Yaskawa INFORM job: DEMO_ROOF_UPPER_0625_3PAINT_32.JBI

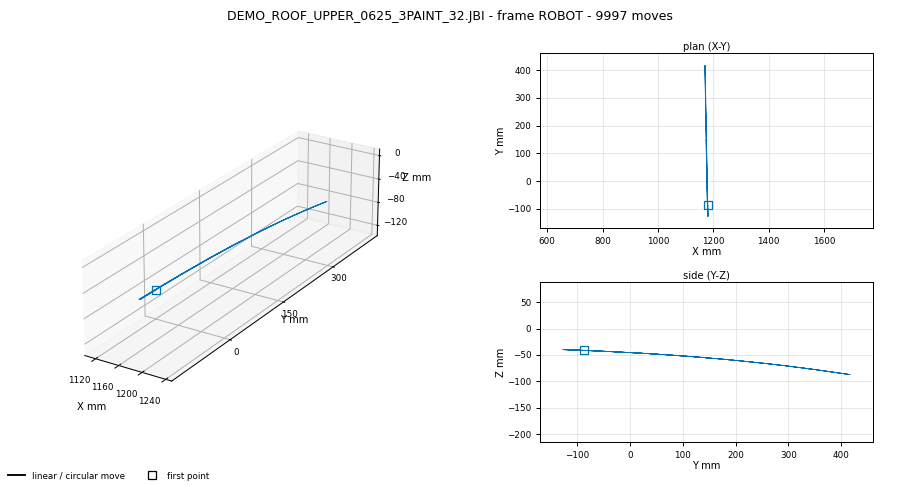
[picture p0: tool path of DEMO_ROOF_UPPER_0625_3PAINT_32.JBI in frame ROBOT, 9997 of 9997 moves have a stored position in this frame; points joined in program order, loops and branches not executed]
/JOB
//NAME DEMO_ROOF_UPPER_0625_3PAINT32
//POS
///NPOS 9997,0,0,0,0,0
///TOOL 0
///USER 0
///POSTYPE ROBOT
///RECTAN
///RCONF 1,0,0,0,0,0,0,0,0,0,0,0,0,0,0,0,0,0,0,0,0,0,0,0
C00000=1180.543,-86.813,-41.166,179.183,5.706,149.254
C00001=1180.548,-87.062,-41.157,179.181,5.706,149.255
C00002=1180.554,-87.312,-41.146,179.179,5.706,149.256
C00003=1180.559,-87.563,-41.136,179.177,5.705,149.256
C00004=1180.565,-87.812,-41.126,179.174,5.706,149.257
C00005=1180.570,-88.062,-41.116,179.172,5.705,149.257
C00006=1180.574,-88.312,-41.106,179.170,5.705,149.258
C00007=1180.580,-88.561,-41.096,179.168,5.704,149.259
C00008=1180.586,-88.811,-41.086,179.165,5.704,149.259
C00009=1180.591,-89.061,-41.075,179.163,5.704,149.260
C00010=1180.596,-89.310,-41.065,179.161,5.704,149.260
C00011=1180.601,-89.560,-41.055,179.159,5.704,149.261
C00012=1180.607,-89.809,-41.045,179.157,5.703,149.262
C00013=1180.612,-90.060,-41.035,179.154,5.703,149.262
C00014=1180.617,-90.310,-41.026,179.153,5.703,149.263
C00015=1180.622,-90.559,-41.015,179.150,5.702,149.264
C00016=1180.627,-90.809,-41.005,179.148,5.703,149.264
C00017=1180.633,-91.059,-40.995,179.146,5.702,149.265
C00018=1180.638,-91.308,-40.985,179.143,5.703,149.265
C00019=1180.644,-91.558,-40.975,179.141,5.702,149.266
C00020=1180.649,-91.809,-40.965,179.139,5.701,149.267
C00021=1180.654,-92.058,-40.955,179.137,5.701,149.267
C00022=1180.659,-92.307,-40.945,179.134,5.701,149.268
C00023=1180.665,-92.557,-40.935,179.132,5.701,149.269
C00024=1180.669,-92.807,-40.925,179.130,5.701,149.269
C00025=1180.675,-93.057,-40.915,179.127,5.700,149.270
C00026=1180.681,-93.307,-40.905,179.126,5.700,149.270
C00027=1180.686,-93.556,-40.896,179.123,5.700,149.271
C00028=1180.691,-93.806,-40.885,179.122,5.700,149.271
C00029=1180.696,-94.056,-40.876,179.119,5.699,149.272
C00030=1180.701,-94.305,-40.866,179.117,5.699,149.273
C00031=1180.707,-94.555,-40.856,179.115,5.699,149.273
C00032=1180.712,-94.804,-40.845,179.112,5.699,149.274
C00033=1180.717,-95.055,-40.836,179.110,5.699,149.275
C00034=1180.723,-95.305,-40.826,179.108,5.698,149.275
C00035=1180.728,-95.554,-40.816,179.106,5.698,149.276
C00036=1180.733,-95.803,-40.806,179.103,5.698,149.276
C00037=1180.739,-96.054,-40.797,179.102,5.698,149.277
C00038=1180.744,-96.304,-40.786,179.099,5.697,149.278
C00039=1180.749,-96.553,-40.777,179.097,5.697,149.278
C00040=1180.755,-96.803,-40.767,179.095,5.697,149.279
C00041=1180.760,-97.052,-40.757,179.092,5.697,149.280
C00042=1180.765,-97.302,-40.747,179.091,5.697,149.280
C00043=1180.771,-97.553,-40.737,179.088,5.696,149.281
C00044=1180.775,-97.802,-40.728,179.086,5.696,149.281
C00045=1180.781,-98.052,-40.718,179.084,5.696,149.282
C00046=1180.786,-98.301,-40.709,179.081,5.695,149.282
C00047=1180.792,-98.551,-40.698,179.079,5.696,149.283
C00048=1180.797,-98.800,-40.688,179.077,5.695,149.284
C00049=1180.802,-99.051,-40.679,179.075,5.695,149.284
C00050=1180.808,-99.301,-40.669,179.073,5.694,149.285
C00051=1180.813,-99.550,-40.660,179.071,5.695,149.285
C00052=1180.818,-99.800,-40.650,179.069,5.694,149.286
C00053=1180.823,-100.049,-40.640,179.066,5.694,149.287
C00054=1180.829,-100.299,-40.631,179.064,5.694,149.287
C00055=1180.834,-100.549,-40.621,179.062,5.693,149.288
C00056=1180.839,-100.799,-40.611,179.060,5.694,149.289
C00057=1180.844,-101.049,-40.601,179.057,5.693,149.289
C00058=1180.850,-101.298,-40.591,179.055,5.693,149.290
C00059=1180.855,-101.570,-40.581,179.053,5.692,149.290
C00060=1180.861,-101.841,-40.571,179.050,5.692,149.291
C00061=1180.868,-102.114,-40.560,179.048,5.692,149.292
C00062=1180.873,-102.385,-40.549,179.046,5.692,149.292
C00063=1180.879,-102.635,-40.540,179.043,5.691,149.293
C00064=1180.883,-102.884,-40.530,179.041,5.692,149.294
C00065=1180.889,-103.134,-40.521,179.039,5.691,149.294
C00066=1180.894,-103.384,-40.511,179.037,5.691,149.295
C00067=1180.899,-103.634,-40.502,179.035,5.691,149.295
C00068=1180.904,-103.884,-40.492,179.033,5.691,149.296
C00069=1180.910,-104.134,-40.483,179.031,5.690,149.297
C00070=1180.915,-104.383,-40.473,179.029,5.691,149.297
C00071=1180.920,-104.633,-40.464,179.026,5.690,149.298
C00072=1180.926,-104.883,-40.453,179.024,5.689,149.298
C00073=1180.931,-105.132,-40.445,179.022,5.689,149.299
C00074=1180.937,-105.383,-40.435,179.019,5.689,149.300
C00075=1180.942,-105.632,-40.425,179.018,5.689,149.300
C00076=1180.947,-105.882,-40.417,179.015,5.689,149.301
C00077=1180.953,-106.131,-40.406,179.014,5.689,149.301
C00078=1180.957,-106.382,-40.397,179.011,5.688,149.302
C00079=1180.963,-106.631,-40.387,179.009,5.688,149.303
C00080=1180.968,-106.881,-40.378,179.007,5.688,149.303
C00081=1180.974,-107.131,-40.368,179.005,5.688,149.304
C00082=1180.979,-107.381,-40.359,179.002,5.688,149.304
C00083=1180.984,-107.630,-40.350,179.001,5.688,149.305
C00084=1180.989,-107.880,-40.340,178.998,5.687,149.306
C00085=1180.995,-108.130,-40.331,178.996,5.686,149.306
C00086=1181.000,-108.380,-40.322,178.994,5.687,149.307
C00087=1181.005,-108.629,-40.312,178.992,5.686,149.307
C00088=1181.011,-108.879,-40.303,178.989,5.686,149.308
C00089=1181.016,-109.129,-40.293,178.987,5.686,149.309
C00090=1181.021,-109.378,-40.284,178.985,5.686,149.309
C00091=1181.026,-109.628,-40.275,178.983,5.685,149.310
C00092=1181.032,-109.878,-40.265,178.981,5.686,149.310
C00093=1181.037,-110.128,-40.256,178.979,5.685,149.311
C00094=1181.042,-110.378,-40.247,178.977,5.685,149.312
C00095=1181.048,-110.627,-40.237,178.974,5.685,149.312
C00096=1181.053,-110.877,-40.228,178.972,5.685,149.313
C00097=1181.058,-111.127,-40.219,178.970,5.684,149.313
C00098=1181.064,-111.377,-40.209,178.968,5.685,149.314
C00099=1181.069,-111.626,-40.200,178.966,5.684,149.314
C00100=1181.074,-111.876,-40.191,178.964,5.684,149.315
C00101=1181.080,-112.126,-40.181,178.962,5.683,149.316
C00102=1181.085,-112.375,-40.172,178.960,5.684,149.316
C00103=1181.090,-112.625,-40.163,178.957,5.683,149.317
C00104=1181.096,-112.875,-40.153,178.955,5.683,149.318
C00105=1181.101,-113.125,-40.144,178.953,5.683,149.318
C00106=1181.106,-113.375,-40.135,178.950,5.682,149.319
C00107=1181.111,-113.624,-40.126,178.949,5.682,149.319
C00108=1181.117,-113.875,-40.116,178.946,5.682,149.320
C00109=1181.122,-114.124,-40.108,178.945,5.682,149.320
C00110=1181.128,-114.374,-40.099,178.942,5.682,149.321
C00111=1181.133,-114.624,-40.088,178.940,5.682,149.322
C00112=1181.138,-114.874,-40.080,178.938,5.681,149.322
C00113=1181.143,-115.124,-40.071,178.936,5.681,149.323
C00114=1181.149,-115.373,-40.062,178.934,5.680,149.323
C00115=1181.155,-115.624,-40.052,178.932,5.681,149.324
C00116=1181.159,-115.873,-40.043,178.930,5.680,149.325
C00117=1181.165,-116.123,-40.034,178.927,5.681,149.325
C00118=1181.170,-116.372,-40.025,178.925,5.680,149.326
C00119=1181.176,-116.622,-40.016,178.923,5.680,149.327
C00120=1181.181,-116.872,-40.007,178.921,5.679,149.327
C00121=1181.187,-117.122,-39.998,178.919,5.680,149.328
C00122=1181.191,-117.371,-39.988,178.917,5.679,149.328
C00123=1181.197,-117.621,-39.979,178.915,5.679,149.329
C00124=1181.203,-117.871,-39.970,178.912,5.679,149.329
C00125=1181.208,-118.121,-39.961,178.911,5.679,149.330
C00126=1181.213,-118.371,-39.952,178.908,5.678,149.331
C00127=1181.218,-118.620,-39.943,178.907,5.678,149.331
C00128=1181.223,-118.870,-39.934,178.904,5.678,149.332
C00129=1181.229,-119.120,-39.925,178.902,5.678,149.332
C00130=1181.235,-119.369,-39.916,178.900,5.678,149.333
C00131=1181.240,-119.619,-39.907,178.898,5.678,149.333
C00132=1181.245,-119.869,-39.898,178.895,5.677,149.334
C00133=1181.250,-120.119,-39.889,178.894,5.677,149.335
C00134=1181.255,-120.368,-39.880,178.892,5.676,149.335
C00135=1181.261,-120.619,-39.870,178.889,5.677,149.336
C00136=1181.266,-120.868,-39.862,178.887,5.676,149.336
C00137=1181.271,-121.118,-39.853,178.885,5.677,149.337
C00138=1181.277,-121.368,-39.844,178.883,5.676,149.338
C00139=1181.282,-121.617,-39.835,178.881,5.676,149.338
C00140=1181.288,-121.867,-39.826,178.879,5.675,149.339
C00141=1181.293,-122.117,-39.817,178.877,5.676,149.339
C00142=1181.299,-122.367,-39.808,178.874,5.675,149.340
C00143=1181.304,-122.617,-39.799,178.873,5.675,149.340
C00144=1181.309,-122.867,-39.790,178.870,5.675,149.341
C00145=1181.314,-123.117,-39.781,178.869,5.675,149.342
C00146=1181.320,-123.366,-39.773,178.866,5.674,149.342
C00147=1181.325,-123.616,-39.764,178.864,5.674,149.343
C00148=1181.330,-123.866,-39.755,178.862,5.675,149.344
C00149=1181.335,-124.115,-39.746,178.860,5.674,149.344
C00150=1181.341,-124.365,-39.737,178.858,5.674,149.345
C00151=1181.346,-124.615,-39.728,178.856,5.674,149.345
C00152=1181.351,-124.865,-39.719,178.854,5.674,149.346
C00153=1181.357,-125.114,-39.710,178.851,5.673,149.346
C00154=1181.363,-125.364,-39.701,178.850,5.673,149.347
C00155=1181.368,-125.614,-39.692,178.847,5.673,149.348
C00156=1181.373,-125.864,-39.684,178.846,5.673,149.348
C00157=1181.378,-126.114,-39.675,178.843,5.672,149.349
C00158=1181.384,-126.363,-39.666,178.841,5.673,149.349
C00159=1181.389,-126.613,-39.658,178.839,5.672,149.350
C00160=1181.394,-126.863,-39.649,178.837,5.672,149.351
C00161=1181.400,-127.113,-39.640,178.835,5.672,149.351
C00162=1181.405,-127.363,-39.631,178.833,5.672,149.352
C00163=1180.984,-127.374,-39.672,178.829,5.675,149.353
C00164=1180.979,-127.124,-39.681,178.831,5.675,149.353
C00165=1180.973,-126.875,-39.689,178.833,5.676,149.352
C00166=1180.967,-126.624,-39.697,178.835,5.675,149.352
C00167=1180.962,-126.374,-39.706,178.837,5.676,149.351
C00168=1180.957,-126.124,-39.715,178.839,5.675,149.351
C00169=1180.952,-125.874,-39.724,178.842,5.676,149.350
C00170=1180.946,-125.625,-39.733,178.843,5.676,149.350
C00171=1180.941,-125.376,-39.741,178.846,5.677,149.349
C00172=1180.936,-125.126,-39.750,178.847,5.677,149.348
C00173=1180.931,-124.876,-39.759,178.850,5.677,149.348
C00174=1180.925,-124.626,-39.768,178.852,5.677,149.347
C00175=1180.920,-124.376,-39.777,178.854,5.678,149.347
C00176=1180.914,-124.127,-39.786,178.856,5.677,149.346
C00177=1180.909,-123.877,-39.795,178.858,5.678,149.345
C00178=1180.903,-123.627,-39.804,178.860,5.678,149.345
C00179=1180.898,-123.377,-39.813,178.863,5.678,149.344
C00180=1180.893,-123.127,-39.822,178.865,5.678,149.344
C00181=1180.888,-122.877,-39.831,178.867,5.679,149.343
C00182=1180.883,-122.628,-39.840,178.868,5.679,149.343
C00183=1180.877,-122.378,-39.848,178.871,5.679,149.342
C00184=1180.872,-122.129,-39.857,178.873,5.679,149.341
C00185=1180.867,-121.879,-39.866,178.875,5.679,149.341
C00186=1180.861,-121.629,-39.875,178.877,5.679,149.340
C00187=1180.856,-121.379,-39.884,178.880,5.680,149.339
C00188=1180.850,-121.129,-39.893,178.881,5.680,149.339
C00189=1180.845,-120.879,-39.902,178.883,5.681,149.338
C00190=1180.839,-120.630,-39.911,178.886,5.680,149.338
C00191=1180.834,-120.380,-39.919,178.888,5.681,149.337
C00192=1180.829,-120.130,-39.928,178.890,5.680,149.337
C00193=1180.823,-119.880,-39.938,178.892,5.681,149.336
C00194=1180.818,-119.630,-39.947,178.894,5.681,149.335
C00195=1180.813,-119.380,-39.956,178.896,5.682,149.335
C00196=1180.808,-119.130,-39.965,178.898,5.681,149.334
C00197=1180.803,-118.881,-39.973,178.901,5.682,149.334
C00198=1180.798,-118.631,-39.983,178.902,5.682,149.333
C00199=1180.792,-118.381,-39.993,178.905,5.682,149.332
C00200=1180.786,-118.132,-40.001,178.906,5.682,149.332
C00201=1180.781,-117.882,-40.010,178.909,5.683,149.331
C00202=1180.776,-117.632,-40.019,178.911,5.683,149.331
C00203=1180.770,-117.382,-40.028,178.913,5.683,149.330
C00204=1180.765,-117.132,-40.037,178.915,5.683,149.330
C00205=1180.759,-116.882,-40.046,178.918,5.683,149.329
C00206=1180.755,-116.633,-40.056,178.919,5.683,149.328
C00207=1180.749,-116.383,-40.065,178.922,5.684,149.328
C00208=1180.744,-116.133,-40.074,178.924,5.684,149.327
C00209=1180.738,-115.883,-40.083,178.926,5.685,149.327
C00210=1180.733,-115.633,-40.092,178.928,5.684,149.326
C00211=1180.728,-115.384,-40.101,178.930,5.685,149.325
C00212=1180.723,-115.134,-40.110,178.932,5.684,149.325
C00213=1180.717,-114.884,-40.120,178.934,5.685,149.324
C00214=1180.711,-114.635,-40.129,178.936,5.685,149.324
C00215=1180.706,-114.385,-40.137,178.939,5.686,149.323
C00216=1180.700,-114.135,-40.147,178.941,5.685,149.322
C00217=1180.696,-113.886,-40.157,178.943,5.686,149.322
C00218=1180.690,-113.636,-40.165,178.945,5.686,149.321
C00219=1180.685,-113.386,-40.174,178.947,5.686,149.321
C00220=1180.679,-113.136,-40.184,178.949,5.686,149.320
C00221=1180.674,-112.887,-40.193,178.951,5.687,149.319
C00222=1180.669,-112.637,-40.202,178.953,5.686,149.319
C00223=1180.663,-112.387,-40.212,178.956,5.687,149.318
C00224=1180.658,-112.137,-40.221,178.957,5.687,149.318
C00225=1180.653,-111.888,-40.230,178.960,5.687,149.317
C00226=1180.648,-111.638,-40.239,178.962,5.687,149.317
C00227=1180.642,-111.388,-40.249,178.964,5.688,149.316
C00228=1180.637,-111.138,-40.258,178.966,5.688,149.315
C00229=1180.632,-110.889,-40.267,178.968,5.688,149.315
C00230=1180.626,-110.638,-40.277,178.970,5.688,149.314
C00231=1180.621,-110.389,-40.286,178.973,5.689,149.313
C00232=1180.616,-110.139,-40.295,178.974,5.689,149.313
C00233=1180.610,-109.889,-40.305,178.977,5.689,149.312
C00234=1180.605,-109.639,-40.314,178.979,5.690,149.312
C00235=1180.600,-109.390,-40.324,178.981,5.689,149.311
C00236=1180.594,-109.140,-40.333,178.984,5.690,149.311
C00237=1180.589,-108.890,-40.342,178.986,5.690,149.310
C00238=1180.584,-108.641,-40.352,178.988,5.690,149.309
C00239=1180.579,-108.391,-40.361,178.990,5.690,149.309
C00240=1180.573,-108.141,-40.370,178.992,5.691,149.308
C00241=1180.568,-107.891,-40.380,178.994,5.690,149.307
C00242=1180.563,-107.641,-40.389,178.996,5.691,149.307
C00243=1180.557,-107.392,-40.399,178.998,5.691,149.306
C00244=1180.552,-107.141,-40.408,179.001,5.692,149.306
C00245=1180.547,-106.891,-40.417,179.003,5.691,149.305
C00246=1180.542,-106.642,-40.427,179.005,5.692,149.305
C00247=1180.536,-106.392,-40.436,179.007,5.691,149.304
C00248=1180.531,-106.143,-40.446,179.009,5.692,149.303
C00249=1180.526,-105.893,-40.455,179.012,5.693,149.303
C00250=1180.521,-105.643,-40.465,179.013,5.693,149.302
C00251=1180.515,-105.393,-40.474,179.016,5.693,149.301
C00252=1180.510,-105.143,-40.483,179.018,5.693,149.301
C00253=1180.504,-104.894,-40.494,179.020,5.693,149.300
C00254=1180.499,-104.644,-40.502,179.022,5.693,149.300
C00255=1180.493,-104.394,-40.513,179.025,5.694,149.299
C00256=1180.488,-104.145,-40.522,179.026,5.694,149.299
C00257=1180.483,-103.894,-40.532,179.029,5.694,149.298
C00258=1180.478,-103.645,-40.541,179.031,5.694,149.297
C00259=1180.473,-103.395,-40.551,179.033,5.695,149.297
C00260=1180.467,-103.145,-40.560,179.035,5.695,149.296
C00261=1180.462,-102.896,-40.570,179.037,5.695,149.295
C00262=1180.457,-102.646,-40.579,179.040,5.696,149.295
C00263=1180.452,-102.397,-40.589,179.042,5.695,149.294
C00264=1180.445,-102.124,-40.600,179.044,5.696,149.294
C00265=1180.440,-101.852,-40.610,179.047,5.696,149.293
C00266=1180.434,-101.582,-40.620,179.049,5.696,149.292
C00267=1180.429,-101.310,-40.631,179.051,5.696,149.292
C00268=1180.423,-101.060,-40.640,179.053,5.696,149.291
C00269=1180.419,-100.810,-40.650,179.056,5.697,149.290
C00270=1180.413,-100.560,-40.660,179.058,5.698,149.290
C00271=1180.407,-100.310,-40.670,179.060,5.697,149.289
C00272=1180.402,-100.061,-40.679,179.063,5.698,149.289
C00273=1180.396,-99.811,-40.689,179.064,5.698,149.288
C00274=1180.391,-99.561,-40.699,179.067,5.698,149.287
C00275=1180.386,-99.312,-40.709,179.068,5.698,149.287
C00276=1180.381,-99.061,-40.718,179.071,5.698,149.286
C00277=1180.376,-98.812,-40.728,179.073,5.699,149.286
C00278=1180.370,-98.562,-40.737,179.075,5.699,149.285
C00279=1180.365,-98.312,-40.747,179.078,5.699,149.284
C00280=1180.359,-98.063,-40.758,179.080,5.699,149.284
C00281=1180.354,-97.813,-40.766,179.082,5.700,149.283
C00282=1180.349,-97.563,-40.777,179.084,5.699,149.283
C00283=1180.344,-97.314,-40.787,179.086,5.700,149.282
C00284=1180.338,-97.063,-40.796,179.088,5.700,149.281
C00285=1180.333,-96.814,-40.806,179.090,5.701,149.281
C00286=1180.328,-96.565,-40.816,179.093,5.701,149.280
C00287=1180.322,-96.314,-40.825,179.095,5.701,149.279
C00288=1180.318,-96.064,-40.835,179.097,5.701,149.279
C00289=1180.312,-95.815,-40.846,179.099,5.701,149.278
C00290=1180.306,-95.565,-40.855,179.102,5.702,149.278
C00291=1180.301,-95.316,-40.865,179.104,5.701,149.277
C00292=1180.296,-95.066,-40.875,179.106,5.702,149.277
C00293=1180.291,-94.816,-40.886,179.109,5.703,149.276
C00294=1180.286,-94.566,-40.894,179.110,5.703,149.275
C00295=1180.280,-94.316,-40.905,179.113,5.703,149.275
C00296=1180.275,-94.067,-40.914,179.114,5.703,149.274
C00297=1180.270,-93.816,-40.924,179.117,5.703,149.273
C00298=1180.264,-93.567,-40.934,179.120,5.704,149.273
C00299=1180.259,-93.317,-40.944,179.121,5.704,149.272
C00300=1180.254,-93.068,-40.954,179.124,5.704,149.272
C00301=1180.248,-92.818,-40.964,179.126,5.704,149.271
C00302=1180.244,-92.568,-40.974,179.128,5.705,149.270
C00303=1180.238,-92.318,-40.984,179.130,5.705,149.270
C00304=1180.232,-92.069,-40.994,179.133,5.705,149.269
C00305=1180.227,-91.819,-41.004,179.135,5.706,149.269
C00306=1180.223,-91.569,-41.014,179.137,5.705,149.268
C00307=1180.217,-91.319,-41.024,179.140,5.706,149.267
C00308=1180.211,-91.070,-41.034,179.141,5.706,149.267
C00309=1180.206,-90.820,-41.044,179.144,5.706,149.266
C00310=1180.201,-90.570,-41.054,179.146,5.707,149.266
C00311=1180.196,-90.321,-41.064,179.148,5.706,149.265
C00312=1180.190,-90.071,-41.075,179.150,5.707,149.264
C00313=1180.185,-89.820,-41.084,179.152,5.707,149.264
C00314=1180.180,-89.571,-41.094,179.155,5.707,149.263
C00315=1180.174,-89.321,-41.104,179.157,5.708,149.263
C00316=1180.169,-89.072,-41.114,179.159,5.708,149.262
C00317=1180.164,-88.822,-41.124,179.162,5.708,149.261
C00318=1180.159,-88.572,-41.135,179.164,5.708,149.261
C00319=1180.153,-88.323,-41.145,179.166,5.709,149.260
C00320=1180.148,-88.073,-41.155,179.168,5.709,149.259
C00321=1180.143,-87.823,-41.165,179.171,5.709,149.259
C00322=1180.138,-87.574,-41.175,179.173,5.710,149.258
C00323=1180.132,-87.323,-41.185,179.175,5.709,149.258
C00324=1180.127,-87.073,-41.195,179.177,5.710,149.257
C00325=1180.122,-86.824,-41.205,179.180,5.710,149.256
C00326=1180.117,-86.574,-41.215,179.181,5.710,149.256
C00327=1180.111,-86.324,-41.226,179.184,5.711,149.255
C00328=1180.106,-86.075,-41.236,179.186,5.710,149.254
C00329=1180.101,-85.825,-41.246,179.188,5.711,149.254
C00330=1180.096,-85.575,-41.256,179.191,5.712,149.253
C00331=1180.090,-85.326,-41.266,179.192,5.712,149.253
C00332=1180.085,-85.076,-41.277,179.195,5.712,149.252
C00333=1180.080,-84.826,-41.287,179.197,5.712,149.252
C00334=1180.074,-84.576,-41.297,179.199,5.712,149.251
C00335=1180.069,-84.326,-41.308,179.202,5.713,149.250
C00336=1180.064,-84.077,-41.317,179.204,5.713,149.250
C00337=1180.059,-83.827,-41.328,179.206,5.713,149.249
C00338=1180.054,-83.577,-41.338,179.208,5.713,149.248
C00339=1180.048,-83.328,-41.348,179.211,5.714,149.248
C00340=1180.042,-83.078,-41.359,179.213,5.714,149.247
C00341=1180.037,-82.828,-41.369,179.215,5.714,149.247
C00342=1180.032,-82.578,-41.379,179.218,5.714,149.246
C00343=1180.027,-82.329,-41.391,179.220,5.715,149.245
C00344=1180.022,-82.079,-41.400,179.222,5.715,149.245
C00345=1180.017,-81.830,-41.411,179.225,5.715,149.244
C00346=1180.012,-81.580,-41.421,179.226,5.715,149.243
C00347=1180.006,-81.330,-41.431,179.229,5.716,149.243
C00348=1180.001,-81.080,-41.442,179.231,5.716,149.242
C00349=1179.996,-80.830,-41.452,179.233,5.716,149.242
C00350=1179.990,-80.581,-41.462,179.235,5.717,149.241
C00351=1179.985,-80.331,-41.473,179.238,5.717,149.240
C00352=1179.979,-80.081,-41.483,179.240,5.717,149.240
C00353=1179.975,-79.831,-41.494,179.242,5.718,149.239
C00354=1179.969,-79.582,-41.505,179.244,5.717,149.238
C00355=1179.963,-79.332,-41.515,179.246,5.718,149.238
C00356=1179.959,-79.082,-41.525,179.249,5.718,149.237
C00357=1179.954,-78.833,-41.535,179.251,5.718,149.237
C00358=1179.949,-78.583,-41.546,179.253,5.719,149.236
C00359=1179.943,-78.334,-41.557,179.256,5.719,149.235
C00360=1179.938,-78.083,-41.567,179.258,5.719,149.235
C00361=1179.933,-77.834,-41.577,179.260,5.720,149.234
C00362=1179.927,-77.584,-41.588,179.263,5.720,149.233
C00363=1179.922,-77.334,-41.598,179.265,5.720,149.233
C00364=1179.917,-77.085,-41.609,179.267,5.720,149.232
C00365=1179.912,-76.835,-41.620,179.269,5.721,149.232
C00366=1179.906,-76.585,-41.630,179.272,5.721,149.231
C00367=1179.901,-76.335,-41.640,179.274,5.721,149.230
C00368=1179.895,-76.065,-41.652,179.277,5.722,149.230
C00369=1179.889,-75.793,-41.664,179.278,5.722,149.229
C00370=1179.884,-75.522,-41.675,179.281,5.722,149.229
C00371=1179.878,-75.252,-41.687,179.284,5.722,149.228
C00372=1179.873,-75.001,-41.697,179.287,5.723,149.227
C00373=1179.867,-74.752,-41.707,179.288,5.723,149.227
C00374=1179.862,-74.502,-41.719,179.291,5.723,149.226
C00375=1179.857,-74.253,-41.729,179.293,5.724,149.225
C00376=1179.852,-74.002,-41.739,179.295,5.724,149.225
C00377=1179.847,-73.754,-41.750,179.298,5.724,149.224
C00378=1179.842,-73.503,-41.761,179.300,5.725,149.224
C00379=1179.836,-73.254,-41.771,179.302,5.725,149.223
C00380=1179.831,-73.004,-41.782,179.305,5.725,149.222
C00381=1179.826,-72.755,-41.793,179.306,5.725,149.222
C00382=1179.820,-72.504,-41.804,179.309,5.725,149.221
C00383=1179.815,-72.255,-41.815,179.311,5.726,149.220
C00384=1179.810,-72.005,-41.825,179.313,5.726,149.220
C00385=1179.804,-71.755,-41.836,179.316,5.726,149.219
C00386=1179.799,-71.506,-41.847,179.318,5.727,149.219
C00387=1179.794,-71.256,-41.857,179.320,5.727,149.218
C00388=1179.789,-71.006,-41.868,179.322,5.727,149.217
C00389=1179.783,-70.757,-41.879,179.325,5.728,149.217
C00390=1179.778,-70.507,-41.889,179.327,5.727,149.216
C00391=1179.772,-70.258,-41.901,179.329,5.728,149.215
C00392=1179.767,-70.007,-41.911,179.332,5.729,149.215
C00393=1179.762,-69.758,-41.921,179.334,5.728,149.214
C00394=1179.757,-69.508,-41.933,179.336,5.729,149.214
C00395=1179.752,-69.258,-41.943,179.339,5.729,149.213
C00396=1179.747,-69.009,-41.954,179.340,5.729,149.212
C00397=1179.742,-68.759,-41.965,179.343,5.730,149.212
C00398=1179.736,-68.509,-41.976,179.346,5.730,149.211
C00399=1179.731,-68.259,-41.987,179.348,5.731,149.210
C00400=1179.726,-68.010,-41.998,179.350,5.731,149.210
C00401=1179.721,-67.760,-42.008,179.353,5.731,149.209
C00402=1179.716,-67.510,-42.020,179.355,5.732,149.209
C00403=1179.709,-67.261,-42.030,179.357,5.732,149.208
C00404=1179.705,-67.011,-42.042,179.359,5.732,149.207
C00405=1179.699,-66.761,-42.052,179.362,5.733,149.207
C00406=1179.694,-66.512,-42.063,179.364,5.732,149.206
C00407=1179.689,-66.262,-42.073,179.366,5.733,149.206
C00408=1179.683,-66.012,-42.085,179.369,5.734,149.205
C00409=1179.678,-65.762,-42.096,179.371,5.733,149.204
C00410=1179.673,-65.513,-42.107,179.373,5.734,149.204
C00411=1179.668,-65.263,-42.117,179.376,5.734,149.203
C00412=1179.663,-65.013,-42.129,179.378,5.734,149.202
C00413=1179.657,-64.763,-42.140,179.380,5.735,149.202
C00414=1179.652,-64.514,-42.151,179.383,5.735,149.201
C00415=1179.647,-64.265,-42.162,179.384,5.735,149.201
C00416=1179.642,-64.015,-42.172,179.387,5.736,149.200
C00417=1179.637,-63.765,-42.184,179.390,5.736,149.199
C00418=1179.631,-63.515,-42.194,179.392,5.737,149.199
C00419=1179.626,-63.265,-42.206,179.394,5.737,149.198
C00420=1179.621,-63.016,-42.218,179.397,5.737,149.197
C00421=1179.615,-62.766,-42.228,179.399,5.738,149.197
C00422=1179.611,-62.516,-42.239,179.401,5.737,149.196
C00423=1179.606,-62.266,-42.250,179.403,5.738,149.195
C00424=1179.600,-62.017,-42.261,179.406,5.739,149.195
C00425=1179.595,-61.767,-42.272,179.408,5.738,149.194
C00426=1179.590,-61.517,-42.283,179.410,5.739,149.193
C00427=1179.584,-61.268,-42.295,179.413,5.739,149.193
C00428=1179.579,-61.018,-42.306,179.415,5.740,149.192
C00429=1179.574,-60.768,-42.316,179.417,5.740,149.192
C00430=1179.568,-60.519,-42.328,179.419,5.740,149.191
C00431=1179.564,-60.269,-42.339,179.422,5.741,149.190
C00432=1179.559,-60.019,-42.351,179.424,5.741,149.190
C00433=1179.553,-59.770,-42.361,179.426,5.741,149.189
C00434=1179.548,-59.520,-42.373,179.429,5.742,149.189
C00435=1179.543,-59.270,-42.384,179.431,5.742,149.188
C00436=1179.537,-59.020,-42.395,179.433,5.742,149.187
C00437=1179.532,-58.771,-42.406,179.436,5.742,149.187
C00438=1179.527,-58.521,-42.417,179.438,5.743,149.186
C00439=1179.522,-58.271,-42.429,179.440,5.743,149.185
C00440=1179.516,-58.022,-42.439,179.443,5.743,149.185
C00441=1179.512,-57.772,-42.451,179.445,5.744,149.184
C00442=1179.506,-57.522,-42.463,179.448,5.744,149.184
C00443=1179.501,-57.273,-42.473,179.449,5.744,149.183
C00444=1179.496,-57.023,-42.485,179.452,5.745,149.182
C00445=1179.491,-56.773,-42.496,179.455,5.745,149.182
C00446=1179.486,-56.523,-42.507,179.456,5.745,149.181
C00447=1179.480,-56.274,-42.519,179.459,5.746,149.180
C00448=1179.475,-56.025,-42.530,179.462,5.746,149.180
C00449=1179.470,-55.775,-42.542,179.464,5.747,149.179
C00450=1179.465,-55.524,-42.553,179.466,5.747,149.179
C00451=1179.459,-55.275,-42.564,179.469,5.747,149.178
C00452=1179.454,-55.026,-42.575,179.471,5.748,149.177
C00453=1179.449,-54.776,-42.587,179.473,5.748,149.177
C00454=1179.444,-54.526,-42.598,179.476,5.748,149.176
C00455=1179.439,-54.276,-42.610,179.478,5.749,149.176
C00456=1179.433,-54.027,-42.621,179.480,5.749,149.175
C00457=1179.428,-53.778,-42.633,179.482,5.749,149.174
C00458=1179.423,-53.527,-42.644,179.485,5.750,149.174
C00459=1179.418,-53.277,-42.655,179.487,5.750,149.173
C00460=1179.412,-53.028,-42.667,179.490,5.750,149.172
C00461=1179.407,-52.778,-42.678,179.492,5.750,149.172
C00462=1179.402,-52.529,-42.690,179.494,5.751,149.171
C00463=1179.397,-52.279,-42.701,179.497,5.751,149.170
C00464=1179.392,-52.029,-42.713,179.499,5.752,149.170
C00465=1179.386,-51.780,-42.724,179.501,5.752,149.169
C00466=1179.381,-51.530,-42.736,179.504,5.752,149.168
C00467=1179.376,-51.280,-42.747,179.506,5.753,149.168
C00468=1179.371,-51.031,-42.759,179.509,5.753,149.167
C00469=1179.366,-50.781,-42.770,179.511,5.753,149.167
C00470=1179.360,-50.532,-42.782,179.513,5.754,149.166
C00471=1179.356,-50.282,-42.793,179.516,5.754,149.165
C00472=1179.350,-50.011,-42.805,179.518,5.755,149.165
C00473=1179.345,-49.741,-42.818,179.521,5.755,149.164
C00474=1179.338,-49.470,-42.830,179.524,5.755,149.163
C00475=1179.333,-49.200,-42.843,179.525,5.756,149.163
C00476=1179.328,-48.950,-42.855,179.528,5.756,149.162
C00477=1179.323,-48.701,-42.866,179.531,5.756,149.161
C00478=1179.317,-48.451,-42.878,179.533,5.757,149.161
C00479=1179.311,-48.201,-42.890,179.535,5.758,149.160
C00480=1179.307,-47.952,-42.901,179.537,5.757,149.160
C00481=1179.301,-47.702,-42.913,179.540,5.758,149.159
C00482=1179.297,-47.452,-42.924,179.542,5.758,149.158
C00483=1179.291,-47.202,-42.936,179.545,5.759,149.158
C00484=1179.286,-46.953,-42.949,179.547,5.759,149.157
C00485=1179.281,-46.704,-42.960,179.549,5.759,149.156
C00486=1179.275,-46.454,-42.971,179.552,5.760,149.156
C00487=1179.270,-46.204,-42.983,179.554,5.761,149.155
C00488=1179.265,-45.954,-42.995,179.556,5.760,149.155
C00489=1179.260,-45.705,-43.006,179.559,5.761,149.154
C00490=1179.255,-45.455,-43.018,179.561,5.761,149.153
C00491=1179.250,-45.205,-43.030,179.564,5.762,149.153
C00492=1179.245,-44.956,-43.042,179.566,5.762,149.152
C00493=1179.240,-44.706,-43.054,179.568,5.762,149.152
C00494=1179.234,-44.457,-43.065,179.571,5.763,149.151
C00495=1179.228,-44.207,-43.077,179.573,5.763,149.150
C00496=1179.224,-43.957,-43.088,179.575,5.764,149.150
C00497=1179.218,-43.707,-43.100,179.577,5.764,149.149
C00498=1179.213,-43.458,-43.113,179.580,5.764,149.148
C00499=1179.208,-43.208,-43.125,179.582,5.765,149.148
C00500=1179.203,-42.958,-43.136,179.585,5.765,149.147
C00501=1179.198,-42.708,-43.148,179.588,5.766,149.146
C00502=1179.192,-42.459,-43.160,179.589,5.766,149.146
C00503=1179.188,-42.210,-43.172,179.592,5.766,149.145
C00504=1179.182,-41.960,-43.184,179.595,5.767,149.145
C00505=1179.177,-41.710,-43.195,179.597,5.767,149.144
C00506=1179.172,-41.460,-43.207,179.599,5.767,149.143
C00507=1179.167,-41.211,-43.219,179.601,5.768,149.143
C00508=1179.162,-40.961,-43.231,179.604,5.768,149.142
C00509=1179.156,-40.712,-43.243,179.606,5.769,149.141
C00510=1179.150,-40.462,-43.255,179.609,5.769,149.141
C00511=1179.146,-40.213,-43.267,179.611,5.769,149.140
C00512=1179.140,-39.963,-43.279,179.613,5.770,149.140
C00513=1179.135,-39.713,-43.290,179.616,5.770,149.139
C00514=1179.130,-39.463,-43.303,179.619,5.771,149.138
C00515=1179.125,-39.214,-43.314,179.621,5.771,149.138
C00516=1179.120,-38.964,-43.326,179.623,5.771,149.137
C00517=1179.115,-38.715,-43.339,179.626,5.771,149.136
C00518=1179.109,-38.465,-43.351,179.628,5.772,149.136
C00519=1179.104,-38.215,-43.363,179.630,5.773,149.135
C00520=1179.099,-37.966,-43.375,179.633,5.773,149.134
C00521=1179.094,-37.716,-43.386,179.635,5.773,149.134
C00522=1179.089,-37.466,-43.398,179.637,5.774,149.133
C00523=1179.083,-37.216,-43.411,179.640,5.774,149.133
C00524=1179.078,-36.967,-43.423,179.642,5.775,149.132
C00525=1179.073,-36.717,-43.435,179.645,5.775,149.131
C00526=1179.068,-36.468,-43.447,179.647,5.776,149.131
C00527=1179.063,-36.218,-43.459,179.649,5.776,149.130
C00528=1179.058,-35.968,-43.471,179.652,5.776,149.130
C00529=1179.052,-35.718,-43.483,179.654,5.777,149.129
C00530=1179.047,-35.469,-43.496,179.657,5.777,149.128
C00531=1179.042,-35.219,-43.508,179.659,5.778,149.128
C00532=1179.037,-34.970,-43.520,179.661,5.778,149.127
C00533=1179.032,-34.719,-43.532,179.663,5.778,149.127
C00534=1179.027,-34.470,-43.544,179.666,5.779,149.126
C00535=1179.022,-34.220,-43.556,179.669,5.779,149.125
C00536=1179.016,-33.970,-43.568,179.671,5.780,149.125
C00537=1179.011,-33.721,-43.581,179.674,5.780,149.124
C00538=1179.006,-33.471,-43.593,179.676,5.780,149.123
C00539=1179.001,-33.222,-43.605,179.678,5.781,149.123
C00540=1178.995,-32.972,-43.617,179.681,5.781,149.122
C00541=1178.990,-32.722,-43.630,179.683,5.782,149.121
C00542=1178.985,-32.473,-43.642,179.686,5.782,149.121
C00543=1178.980,-32.223,-43.654,179.688,5.783,149.120
C00544=1178.975,-31.974,-43.667,179.690,5.783,149.119
C00545=1178.969,-31.724,-43.679,179.693,5.783,149.119
C00546=1178.964,-31.475,-43.691,179.695,5.784,149.118
C00547=1178.960,-31.224,-43.703,179.698,5.784,149.118
C00548=1178.955,-30.975,-43.716,179.700,5.785,149.117
C00549=1178.949,-30.725,-43.727,179.702,5.786,149.116
C00550=1178.944,-30.476,-43.740,179.705,5.785,149.116
C00551=1178.939,-30.226,-43.753,179.707,5.786,149.115
C00552=1178.934,-29.977,-43.765,179.709,5.787,149.115
C00553=1178.929,-29.727,-43.777,179.712,5.787,149.114
C00554=1178.923,-29.477,-43.789,179.715,5.787,149.113
C00555=1178.919,-29.227,-43.802,179.717,5.788,149.113
C00556=1178.913,-28.978,-43.815,179.719,5.788,149.112
C00557=1178.908,-28.728,-43.826,179.722,5.788,149.111
C00558=1178.903,-28.479,-43.839,179.724,5.789,149.111
C00559=1178.898,-28.229,-43.852,179.726,5.790,149.110
C00560=1178.892,-27.979,-43.864,179.729,5.790,149.109
C00561=1178.887,-27.730,-43.876,179.731,5.791,149.109
C00562=1178.883,-27.480,-43.889,179.734,5.791,149.108
C00563=1178.877,-27.230,-43.901,179.736,5.791,149.108
C00564=1178.871,-26.981,-43.914,179.739,5.791,149.107
C00565=1178.866,-26.731,-43.927,179.741,5.792,149.106
C00566=1178.861,-26.482,-43.939,179.744,5.793,149.106
C00567=1178.856,-26.232,-43.951,179.746,5.793,149.105
C00568=1178.851,-25.982,-43.964,179.748,5.794,149.105
C00569=1178.846,-25.733,-43.977,179.751,5.794,149.104
C00570=1178.841,-25.483,-43.989,179.753,5.794,149.103
C00571=1178.836,-25.233,-44.001,179.755,5.795,149.103
C00572=1178.830,-24.984,-44.014,179.758,5.795,149.102
C00573=1178.826,-24.734,-44.027,179.761,5.796,149.101
C00574=1178.821,-24.485,-44.040,179.763,5.797,149.101
C00575=1178.815,-24.235,-44.051,179.765,5.797,149.100
C00576=1178.810,-23.965,-44.066,179.768,5.798,149.099
C00577=1178.804,-23.696,-44.079,179.771,5.798,149.099
C00578=1178.798,-23.426,-44.093,179.773,5.798,149.098
C00579=1178.793,-23.155,-44.106,179.776,5.799,149.097
C00580=1178.788,-22.906,-44.119,179.778,5.800,149.097
C00581=1178.783,-22.657,-44.131,179.781,5.800,149.096
C00582=1178.778,-22.407,-44.144,179.784,5.801,149.096
C00583=1178.772,-22.158,-44.157,179.785,5.801,149.095
C00584=1178.767,-21.908,-44.170,179.788,5.801,149.094
C00585=1178.762,-21.658,-44.182,179.790,5.802,149.094
C00586=1178.757,-21.408,-44.195,179.793,5.802,149.093
C00587=1178.752,-21.159,-44.207,179.795,5.803,149.092
C00588=1178.746,-20.909,-44.221,179.798,5.803,149.092
C00589=1178.741,-20.659,-44.233,179.800,5.804,149.091
C00590=1178.736,-20.410,-44.246,179.803,5.805,149.091
C00591=1178.731,-20.161,-44.259,179.805,5.805,149.090
C00592=1178.726,-19.911,-44.272,179.808,5.805,149.089
C00593=1178.721,-19.661,-44.285,179.810,5.805,149.089
C00594=1178.715,-19.412,-44.297,179.812,5.806,149.088
C00595=1178.711,-19.162,-44.310,179.815,5.806,149.087
C00596=1178.705,-18.912,-44.322,179.817,5.807,149.087
C00597=1178.700,-18.663,-44.335,179.820,5.808,149.086
C00598=1178.694,-18.413,-44.348,179.823,5.808,149.086
C00599=1178.690,-18.163,-44.361,179.825,5.809,149.085
C00600=1178.685,-17.914,-44.374,179.827,5.809,149.084
C00601=1178.679,-17.664,-44.387,179.830,5.810,149.084
C00602=1178.674,-17.414,-44.400,179.832,5.810,149.083
C00603=1178.669,-17.165,-44.412,179.834,5.810,149.083
C00604=1178.664,-16.915,-44.425,179.837,5.811,149.082
C00605=1178.659,-16.665,-44.439,179.839,5.812,149.081
C00606=1178.654,-16.416,-44.451,179.842,5.812,149.081
C00607=1178.649,-16.166,-44.464,179.844,5.813,149.080
C00608=1178.643,-15.917,-44.478,179.847,5.813,149.079
C00609=1178.639,-15.667,-44.491,179.849,5.814,149.079
C00610=1178.633,-15.418,-44.503,179.852,5.814,149.078
C00611=1178.629,-15.168,-44.516,179.855,5.815,149.077
C00612=1178.623,-14.918,-44.529,179.857,5.816,149.077
C00613=1178.618,-14.669,-44.542,179.859,5.815,149.076
C00614=1178.613,-14.419,-44.555,179.861,5.816,149.076
C00615=1178.608,-14.169,-44.568,179.864,5.817,149.075
C00616=1178.602,-13.920,-44.581,179.866,5.817,149.074
C00617=1178.598,-13.670,-44.594,179.869,5.817,149.074
C00618=1178.592,-13.420,-44.607,179.871,5.818,149.073
C00619=1178.587,-13.172,-44.620,179.874,5.819,149.073
C00620=1178.582,-12.921,-44.634,179.876,5.819,149.072
C00621=1178.577,-12.672,-44.646,179.879,5.820,149.071
C00622=1178.572,-12.422,-44.659,179.881,5.820,149.071
C00623=1178.566,-12.172,-44.673,179.884,5.821,149.070
C00624=1178.561,-11.923,-44.685,179.886,5.822,149.070
C00625=1178.557,-11.674,-44.699,179.889,5.822,149.069
C00626=1178.551,-11.424,-44.712,179.891,5.822,149.068
C00627=1178.546,-11.175,-44.725,179.893,5.823,149.068
C00628=1178.541,-10.924,-44.738,179.896,5.823,149.067
C00629=1178.536,-10.675,-44.751,179.898,5.824,149.066
C00630=1178.532,-10.426,-44.764,179.901,5.824,149.066
C00631=1178.526,-10.176,-44.778,179.903,5.825,149.065
C00632=1178.521,-9.926,-44.791,179.906,5.825,149.064
C00633=1178.515,-9.676,-44.804,179.908,5.826,149.064
C00634=1178.510,-9.428,-44.817,179.911,5.827,149.063
C00635=1178.505,-9.177,-44.831,179.913,5.827,149.063
C00636=1178.500,-8.928,-44.843,179.916,5.828,149.062
C00637=1178.495,-8.678,-44.857,179.918,5.828,149.061
C00638=1178.490,-8.429,-44.870,179.921,5.829,149.061
C00639=1178.485,-8.179,-44.884,179.923,5.829,149.060
C00640=1178.480,-7.929,-44.896,179.926,5.830,149.060
C00641=1178.475,-7.680,-44.910,179.928,5.831,149.059
C00642=1178.470,-7.430,-44.923,179.931,5.831,149.058
C00643=1178.464,-7.181,-44.936,179.933,5.832,149.058
C00644=1178.459,-6.931,-44.950,179.936,5.832,149.057
C00645=1178.454,-6.682,-44.963,179.938,5.832,149.056
C00646=1178.449,-6.432,-44.976,179.940,5.833,149.056
C00647=1178.444,-6.183,-44.990,179.943,5.833,149.055
C00648=1178.439,-5.933,-45.003,179.945,5.834,149.055
C00649=1178.433,-5.683,-45.016,179.947,5.835,149.054
C00650=1178.429,-5.434,-45.030,179.950,5.835,149.053
C00651=1178.423,-5.184,-45.043,179.953,5.836,149.053
C00652=1178.419,-4.935,-45.057,179.955,5.836,149.052
C00653=1178.413,-4.685,-45.070,179.958,5.837,149.052
C00654=1178.408,-4.435,-45.083,179.960,5.837,149.051
C00655=1178.403,-4.186,-45.097,179.963,5.838,149.050
C00656=1178.398,-3.936,-45.110,179.965,5.839,149.050
C00657=1178.393,-3.687,-45.124,179.968,5.839,149.049
C00658=1178.388,-3.437,-45.137,179.970,5.840,149.048
C00659=1178.383,-3.188,-45.151,179.973,5.840,149.048
C00660=1178.377,-2.938,-45.164,179.975,5.841,149.047
C00661=1178.373,-2.689,-45.178,179.978,5.841,149.046
C00662=1178.367,-2.439,-45.191,179.980,5.842,149.046
C00663=1178.362,-2.188,-45.205,179.983,5.843,149.045
C00664=1178.357,-1.940,-45.218,179.985,5.843,149.045
C00665=1178.352,-1.689,-45.232,179.988,5.844,149.044
C00666=1178.347,-1.440,-45.246,179.990,5.844,149.043
C00667=1178.342,-1.191,-45.259,179.993,5.845,149.043
C00668=1178.336,-0.941,-45.272,179.995,5.846,149.042
C00669=1178.332,-0.692,-45.286,179.998,5.846,149.042
C00670=1178.326,-0.442,-45.299,-180.000,5.847,149.041
C00671=1178.321,-0.192,-45.314,-179.998,5.848,149.040
C00672=1178.316,0.057,-45.326,-179.995,5.848,149.040
C00673=1178.311,0.307,-45.340,-179.992,5.848,149.039
C00674=1178.306,0.557,-45.354,-179.990,5.849,149.039
C00675=1178.301,0.806,-45.368,-179.987,5.850,149.038
C00676=1178.296,1.055,-45.382,-179.985,5.850,149.037
C00677=1178.290,1.305,-45.395,-179.983,5.851,149.037
C00678=1178.285,1.555,-45.409,-179.980,5.852,149.036
C00679=1178.281,1.805,-45.422,-179.977,5.852,149.035
C00680=1178.275,2.073,-45.437,-179.975,5.852,149.035
C00681=1178.269,2.343,-45.452,-179.972,5.853,149.034
C00682=1178.264,2.612,-45.467,-179.970,5.854,149.034
C00683=1178.259,2.882,-45.482,-179.967,5.855,149.033
C00684=1178.253,3.131,-45.496,-179.964,5.856,149.032
C00685=1178.249,3.380,-45.509,-179.961,5.856,149.032
C00686=1178.244,3.630,-45.523,-179.959,5.857,149.031
C00687=1178.238,3.879,-45.537,-179.956,5.857,149.030
C00688=1178.233,4.129,-45.551,-179.954,5.858,149.030
C00689=1178.228,4.378,-45.564,-179.952,5.859,149.029
C00690=1178.223,4.628,-45.578,-179.949,5.859,149.029
C00691=1178.218,4.878,-45.592,-179.946,5.860,149.028
C00692=1178.212,5.127,-45.606,-179.944,5.860,149.027
C00693=1178.208,5.377,-45.619,-179.941,5.861,149.027
C00694=1178.203,5.627,-45.633,-179.939,5.861,149.026
C00695=1178.197,5.876,-45.647,-179.937,5.862,149.026
C00696=1178.193,6.125,-45.661,-179.934,5.863,149.025
C00697=1178.187,6.376,-45.675,-179.931,5.863,149.024
C00698=1178.182,6.624,-45.688,-179.929,5.864,149.024
C00699=1178.177,6.874,-45.703,-179.926,5.864,149.023
C00700=1178.173,7.124,-45.717,-179.924,5.865,149.022
C00701=1178.167,7.373,-45.731,-179.922,5.866,149.022
C00702=1178.162,7.623,-45.744,-179.919,5.866,149.021
C00703=1178.157,7.873,-45.759,-179.916,5.867,149.021
C00704=1178.152,8.122,-45.773,-179.914,5.868,149.020
C00705=1178.147,8.371,-45.786,-179.912,5.868,149.019
C00706=1178.142,8.621,-45.801,-179.909,5.869,149.019
C00707=1178.137,8.871,-45.815,-179.907,5.869,149.018
C00708=1178.131,9.120,-45.828,-179.904,5.870,149.018
C00709=1178.126,9.370,-45.842,-179.901,5.870,149.017
C00710=1178.121,9.620,-45.857,-179.899,5.871,149.016
C00711=1178.116,9.869,-45.871,-179.897,5.872,149.016
C00712=1178.111,10.118,-45.885,-179.894,5.872,149.015
C00713=1178.107,10.368,-45.898,-179.892,5.873,149.015
C00714=1178.102,10.617,-45.913,-179.889,5.873,149.014
C00715=1178.096,10.866,-45.927,-179.886,5.875,149.013
C00716=1178.091,11.116,-45.941,-179.884,5.876,149.013
C00717=1178.086,11.366,-45.955,-179.881,5.876,149.012
C00718=1178.081,11.616,-45.969,-179.878,5.877,149.011
C00719=1178.076,11.865,-45.983,-179.876,5.877,149.011
C00720=1178.070,12.115,-45.997,-179.874,5.878,149.010
C00721=1178.065,12.365,-46.011,-179.871,5.878,149.010
C00722=1178.060,12.614,-46.025,-179.869,5.879,149.009
C00723=1178.056,12.864,-46.040,-179.866,5.880,149.008
C00724=1178.050,13.113,-46.054,-179.863,5.880,149.008
C00725=1178.045,13.363,-46.068,-179.861,5.881,149.007
C00726=1178.040,13.613,-46.082,-179.859,5.881,149.007
C00727=1178.035,13.862,-46.097,-179.856,5.882,149.006
C00728=1178.030,14.111,-46.111,-179.854,5.883,149.005
C00729=1178.025,14.360,-46.125,-179.851,5.883,149.005
C00730=1178.020,14.610,-46.140,-179.849,5.884,149.004
C00731=1178.015,14.860,-46.154,-179.846,5.885,149.004
C00732=1178.010,15.109,-46.168,-179.843,5.886,149.003
C00733=1178.005,15.359,-46.183,-179.841,5.886,149.002
C00734=1178.000,15.608,-46.196,-179.838,5.887,149.002
C00735=1177.995,15.858,-46.211,-179.836,5.888,149.001
C00736=1177.990,16.108,-46.225,-179.834,5.889,149.001
C00737=1177.985,16.357,-46.239,-179.831,5.889,149.000
C00738=1177.980,16.607,-46.254,-179.828,5.890,148.999
C00739=1177.974,16.856,-46.267,-179.826,5.890,148.999
C00740=1177.969,17.105,-46.282,-179.823,5.891,148.998
C00741=1177.965,17.355,-46.297,-179.821,5.891,148.997
C00742=1177.960,17.605,-46.311,-179.819,5.892,148.997
C00743=1177.954,17.855,-46.326,-179.815,5.893,148.996
C00744=1177.949,18.104,-46.340,-179.813,5.894,148.996
C00745=1177.944,18.354,-46.354,-179.811,5.895,148.995
C00746=1177.939,18.602,-46.369,-179.808,5.895,148.995
C00747=1177.934,18.852,-46.383,-179.805,5.896,148.994
C00748=1177.929,19.102,-46.398,-179.803,5.897,148.993
C00749=1177.924,19.351,-46.412,-179.800,5.897,148.993
C00750=1177.919,19.601,-46.426,-179.798,5.898,148.992
C00751=1177.914,19.850,-46.441,-179.796,5.898,148.992
C00752=1177.909,20.100,-46.456,-179.793,5.899,148.991
C00753=1177.904,20.350,-46.470,-179.790,5.900,148.990
C00754=1177.899,20.600,-46.485,-179.788,5.901,148.990
C00755=1177.893,20.848,-46.499,-179.785,5.902,148.989
C00756=1177.888,21.098,-46.513,-179.783,5.902,148.989
C00757=1177.883,21.348,-46.528,-179.780,5.903,148.988
C00758=1177.878,21.597,-46.543,-179.777,5.903,148.987
C00759=1177.873,21.847,-46.558,-179.775,5.904,148.987
C00760=1177.868,22.096,-46.572,-179.773,5.905,148.986
C00761=1177.863,22.346,-46.586,-179.770,5.905,148.985
C00762=1177.859,22.595,-46.601,-179.767,5.907,148.985
C00763=1177.853,22.845,-46.616,-179.765,5.907,148.984
C00764=1177.848,23.095,-46.630,-179.762,5.908,148.984
C00765=1177.843,23.344,-46.645,-179.760,5.909,148.983
C00766=1177.838,23.594,-46.660,-179.757,5.909,148.983
C00767=1177.834,23.843,-46.675,-179.755,5.910,148.982
C00768=1177.827,24.092,-46.689,-179.752,5.911,148.981
C00769=1177.822,24.342,-46.703,-179.750,5.911,148.981
C00770=1177.818,24.591,-46.718,-179.748,5.912,148.980
C00771=1177.813,24.841,-46.733,-179.744,5.913,148.980
C00772=1177.807,25.090,-46.748,-179.742,5.914,148.979
C00773=1177.802,25.340,-46.763,-179.740,5.915,148.978
C00774=1177.798,25.589,-46.777,-179.737,5.915,148.978
C00775=1177.792,25.839,-46.792,-179.734,5.915,148.977
C00776=1177.787,26.089,-46.807,-179.732,5.916,148.977
C00777=1177.783,26.338,-46.822,-179.729,5.917,148.976
C00778=1177.778,26.587,-46.836,-179.726,5.918,148.975
C00779=1177.772,26.837,-46.852,-179.724,5.919,148.975
C00780=1177.767,27.086,-46.866,-179.721,5.919,148.974
C00781=1177.763,27.336,-46.881,-179.719,5.920,148.974
C00782=1177.757,27.586,-46.896,-179.717,5.921,148.973
C00783=1177.752,27.835,-46.911,-179.714,5.921,148.972
C00784=1177.747,28.103,-46.926,-179.711,5.923,148.972
C00785=1177.741,28.373,-46.943,-179.709,5.923,148.971
C00786=1177.736,28.641,-46.958,-179.706,5.924,148.971
C00787=1177.730,28.910,-46.975,-179.703,5.925,148.970
C00788=1177.726,29.160,-46.990,-179.700,5.926,148.969
C00789=1177.721,29.409,-47.004,-179.698,5.927,148.969
C00790=1177.715,29.659,-47.020,-179.695,5.927,148.968
C00791=1177.710,29.908,-47.034,-179.693,5.928,148.967
C00792=1177.705,30.158,-47.049,-179.690,5.928,148.967
C00793=1177.700,30.407,-47.064,-179.688,5.929,148.966
C00794=1177.695,30.657,-47.079,-179.685,5.931,148.966
C00795=1177.691,30.907,-47.095,-179.682,5.931,148.965
C00796=1177.686,31.156,-47.109,-179.680,5.932,148.964
C00797=1177.680,31.406,-47.124,-179.678,5.932,148.964
C00798=1177.676,31.655,-47.139,-179.675,5.933,148.963
C00799=1177.671,31.905,-47.154,-179.672,5.933,148.963
C00800=1177.665,32.154,-47.169,-179.670,5.935,148.962
C00801=1177.661,32.403,-47.184,-179.667,5.936,148.962
C00802=1177.655,32.653,-47.199,-179.665,5.936,148.961
C00803=1177.650,32.902,-47.214,-179.662,5.937,148.960
C00804=1177.645,33.152,-47.230,-179.659,5.937,148.960
C00805=1177.640,33.401,-47.244,-179.657,5.939,148.959
C00806=1177.635,33.651,-47.260,-179.654,5.940,148.959
C00807=1177.630,33.901,-47.275,-179.651,5.940,148.958
C00808=1177.625,34.150,-47.291,-179.649,5.941,148.957
C00809=1177.620,34.400,-47.305,-179.647,5.941,148.957
C00810=1177.615,34.649,-47.320,-179.644,5.942,148.956
C00811=1177.610,34.898,-47.335,-179.641,5.944,148.956
C00812=1177.605,35.148,-47.351,-179.639,5.944,148.955
C00813=1177.600,35.397,-47.365,-179.636,5.945,148.955
C00814=1177.594,35.647,-47.381,-179.634,5.946,148.954
C00815=1177.590,35.896,-47.396,-179.632,5.946,148.953
C00816=1177.585,36.146,-47.412,-179.628,5.948,148.953
C00817=1177.580,36.396,-47.426,-179.626,5.948,148.952
C00818=1177.575,36.645,-47.442,-179.624,5.949,148.952
C00819=1177.570,36.894,-47.457,-179.621,5.950,148.951
C00820=1177.565,37.143,-47.472,-179.618,5.950,148.950
C00821=1177.560,37.394,-47.488,-179.616,5.952,148.950
C00822=1177.555,37.643,-47.503,-179.613,5.952,148.949
C00823=1177.550,37.892,-47.519,-179.611,5.953,148.949
C00824=1177.545,38.142,-47.533,-179.608,5.954,148.948
C00825=1177.539,38.391,-47.549,-179.605,5.954,148.947
C00826=1177.534,38.641,-47.564,-179.603,5.956,148.947
C00827=1177.530,38.890,-47.580,-179.600,5.956,148.946
C00828=1177.525,39.140,-47.595,-179.598,5.957,148.946
C00829=1177.520,39.389,-47.610,-179.595,5.958,148.945
C00830=1177.515,39.638,-47.626,-179.593,5.958,148.944
C00831=1177.509,39.888,-47.641,-179.590,5.960,148.944
C00832=1177.505,40.137,-47.657,-179.587,5.960,148.943
C00833=1177.500,40.387,-47.672,-179.585,5.961,148.943
C00834=1177.494,40.636,-47.688,-179.582,5.962,148.942
C00835=1177.490,40.885,-47.703,-179.579,5.963,148.942
C00836=1177.484,41.135,-47.719,-179.577,5.964,148.941
C00837=1177.479,41.385,-47.734,-179.574,5.964,148.940
C00838=1177.475,41.635,-47.749,-179.572,5.965,148.940
C00839=1177.469,41.884,-47.764,-179.570,5.966,148.939
C00840=1177.464,42.133,-47.781,-179.566,5.967,148.939
C00841=1177.460,42.383,-47.796,-179.564,5.968,148.938
C00842=1177.455,42.632,-47.812,-179.562,5.968,148.938
C00843=1177.449,42.881,-47.827,-179.559,5.969,148.937
C00844=1177.445,43.130,-47.842,-179.556,5.971,148.936
C00845=1177.440,43.381,-47.858,-179.554,5.971,148.936
C00846=1177.434,43.630,-47.874,-179.551,5.972,148.935
C00847=1177.429,43.879,-47.889,-179.549,5.972,148.935
C00848=1177.425,44.129,-47.905,-179.546,5.974,148.934
C00849=1177.420,44.379,-47.920,-179.543,5.975,148.933
C00850=1177.414,44.628,-47.936,-179.541,5.975,148.933
C00851=1177.409,44.877,-47.951,-179.539,5.976,148.932
C00852=1177.405,45.127,-47.967,-179.535,5.977,148.932
C00853=1177.399,45.377,-47.982,-179.533,5.978,148.931
C00854=1177.394,45.625,-47.999,-179.531,5.979,148.931
C00855=1177.390,45.875,-48.015,-179.528,5.980,148.930
C00856=1177.385,46.125,-48.030,-179.525,5.981,148.929
C00857=1177.379,46.374,-48.045,-179.523,5.981,148.929
C00858=1177.375,46.624,-48.061,-179.520,5.982,148.928
C00859=1177.369,46.873,-48.077,-179.518,5.983,148.928
C00860=1177.364,47.122,-48.093,-179.515,5.984,148.927
C00861=1177.360,47.372,-48.108,-179.512,5.985,148.927
C00862=1177.355,47.621,-48.124,-179.510,5.985,148.926
C00863=1177.349,47.871,-48.140,-179.508,5.986,148.925
C00864=1177.345,48.120,-48.156,-179.504,5.988,148.925
C00865=1177.340,48.370,-48.172,-179.502,5.989,148.924
C00866=1177.334,48.619,-48.187,-179.500,5.989,148.924
C00867=1177.330,48.869,-48.203,-179.497,5.990,148.923
C00868=1177.325,49.118,-48.219,-179.494,5.991,148.923
C00869=1177.320,49.367,-48.235,-179.492,5.992,148.922
C00870=1177.315,49.617,-48.251,-179.489,5.993,148.921
C00871=1177.309,49.867,-48.266,-179.486,5.994,148.921
C00872=1177.305,50.116,-48.283,-179.484,5.995,148.920
C00873=1177.300,50.365,-48.298,-179.481,5.995,148.920
C00874=1177.294,50.615,-48.314,-179.479,5.996,148.919
C00875=1177.290,50.864,-48.330,-179.476,5.997,148.919
C00876=1177.285,51.113,-48.346,-179.473,5.998,148.918
C00877=1177.280,51.364,-48.362,-179.471,5.999,148.917
C00878=1177.275,51.612,-48.378,-179.468,6.000,148.917
C00879=1177.270,51.862,-48.394,-179.466,6.001,148.916
C00880=1177.265,52.112,-48.410,-179.463,6.002,148.916
C00881=1177.260,52.361,-48.426,-179.461,6.002,148.915
C00882=1177.255,52.611,-48.442,-179.458,6.004,148.915
C00883=1177.250,52.859,-48.458,-179.455,6.004,148.914
C00884=1177.245,53.109,-48.474,-179.453,6.005,148.913
C00885=1177.240,53.359,-48.490,-179.450,6.006,148.913
C00886=1177.235,53.608,-48.506,-179.448,6.007,148.912
C00887=1177.230,53.858,-48.522,-179.445,6.008,148.912
C00888=1177.225,54.126,-48.540,-179.442,6.009,148.911
C00889=1177.219,54.394,-48.557,-179.440,6.010,148.911
C00890=1177.214,54.663,-48.574,-179.436,6.011,148.910
C00891=1177.209,54.932,-48.591,-179.434,6.012,148.909
C00892=1177.204,55.181,-48.607,-179.432,6.013,148.909
C00893=1177.199,55.431,-48.623,-179.428,6.014,148.908
C00894=1177.194,55.680,-48.640,-179.426,6.015,148.908
C00895=1177.189,55.930,-48.656,-179.424,6.015,148.907
C00896=1177.184,56.178,-48.672,-179.420,6.017,148.906
C00897=1177.179,56.429,-48.688,-179.418,6.018,148.906
C00898=1177.174,56.677,-48.704,-179.416,6.018,148.905
C00899=1177.169,56.927,-48.720,-179.413,6.020,148.905
C00900=1177.164,57.176,-48.736,-179.410,6.020,148.904
C00901=1177.159,57.426,-48.754,-179.408,6.021,148.904
C00902=1177.154,57.675,-48.769,-179.405,6.023,148.903
C00903=1177.149,57.925,-48.786,-179.403,6.023,148.903
C00904=1177.144,58.174,-48.801,-179.400,6.024,148.902
C00905=1177.139,58.424,-48.818,-179.397,6.025,148.901
C00906=1177.134,58.673,-48.834,-179.395,6.026,148.901
C00907=1177.129,58.923,-48.850,-179.392,6.027,148.900
C00908=1177.124,59.171,-48.867,-179.389,6.028,148.900
C00909=1177.120,59.422,-48.883,-179.387,6.029,148.899
C00910=1177.114,59.671,-48.900,-179.385,6.030,148.899
C00911=1177.109,59.920,-48.916,-179.381,6.031,148.898
C00912=1177.104,60.170,-48.932,-179.379,6.032,148.898
C00913=1177.099,60.419,-48.948,-179.377,6.033,148.897
C00914=1177.095,60.669,-48.965,-179.374,6.034,148.897
C00915=1177.090,60.917,-48.981,-179.371,6.035,148.896
C00916=1177.085,61.167,-48.997,-179.369,6.036,148.895
C00917=1177.079,61.416,-49.014,-179.366,6.037,148.895
C00918=1177.075,61.666,-49.031,-179.363,6.037,148.894
C00919=1177.069,61.915,-49.047,-179.361,6.038,148.894
C00920=1177.065,62.165,-49.063,-179.358,6.040,148.893
C00921=1177.060,62.414,-49.080,-179.356,6.041,148.893
C00922=1177.055,62.663,-49.097,-179.353,6.041,148.892
C00923=1177.050,62.914,-49.113,-179.350,6.043,148.891
C00924=1177.045,63.162,-49.129,-179.348,6.043,148.891
C00925=1177.040,63.412,-49.146,-179.346,6.044,148.890
C00926=1177.036,63.661,-49.162,-179.342,6.045,148.890
C00927=1177.030,63.910,-49.179,-179.340,6.046,148.889
C00928=1177.025,64.160,-49.195,-179.338,6.047,148.889
C00929=1177.020,64.409,-49.212,-179.335,6.049,148.888
C00930=1177.016,64.659,-49.228,-179.332,6.049,148.887
C00931=1177.010,64.909,-49.245,-179.329,6.051,148.887
C00932=1177.005,65.157,-49.262,-179.327,6.051,148.886
C00933=1177.001,65.407,-49.278,-179.325,6.052,148.886
C00934=1176.996,65.657,-49.296,-179.321,6.054,148.885
C00935=1176.990,65.906,-49.311,-179.319,6.054,148.885
C00936=1176.986,66.156,-49.328,-179.317,6.055,148.884
C00937=1176.981,66.405,-49.345,-179.313,6.056,148.884
C00938=1176.975,66.654,-49.362,-179.311,6.057,148.883
C00939=1176.971,66.904,-49.378,-179.308,6.058,148.882
C00940=1176.966,67.153,-49.395,-179.306,6.059,148.882
C00941=1176.961,67.402,-49.412,-179.303,6.060,148.881
C00942=1176.956,67.652,-49.428,-179.301,6.062,148.881
C00943=1176.952,67.901,-49.445,-179.298,6.062,148.880
C00944=1176.946,68.150,-49.462,-179.295,6.064,148.880
C00945=1176.941,68.400,-49.479,-179.293,6.064,148.879
C00946=1176.937,68.649,-49.495,-179.290,6.065,148.879
C00947=1176.931,68.898,-49.512,-179.287,6.067,148.878
C00948=1176.927,69.148,-49.529,-179.285,6.067,148.878
C00949=1176.921,69.398,-49.546,-179.282,6.068,148.877
C00950=1176.917,69.647,-49.563,-179.280,6.070,148.877
C00951=1176.912,69.896,-49.579,-179.277,6.070,148.876
C00952=1176.907,70.146,-49.596,-179.274,6.072,148.875
C00953=1176.902,70.395,-49.613,-179.272,6.072,148.875
C00954=1176.896,70.644,-49.630,-179.270,6.073,148.874
C00955=1176.892,70.894,-49.647,-179.266,6.075,148.874
C00956=1176.887,71.143,-49.663,-179.264,6.076,148.873
C00957=1176.882,71.393,-49.681,-179.261,6.077,148.873
C00958=1176.877,71.641,-49.698,-179.259,6.078,148.872
C00959=1176.872,71.891,-49.715,-179.256,6.079,148.872
C00960=1176.868,72.140,-49.732,-179.254,6.080,148.871
C00961=1176.862,72.390,-49.749,-179.251,6.080,148.870
C00962=1176.857,72.639,-49.765,-179.248,6.082,148.870
C00963=1176.852,72.889,-49.782,-179.246,6.083,148.869
C00964=1176.848,73.138,-49.799,-179.243,6.084,148.869
C00965=1176.843,73.387,-49.817,-179.240,6.085,148.868
C00966=1176.838,73.636,-49.833,-179.238,6.086,148.868
C00967=1176.832,73.886,-49.851,-179.235,6.087,148.867
C00968=1176.828,74.135,-49.867,-179.233,6.088,148.867
C00969=1176.823,74.385,-49.885,-179.229,6.089,148.866
C00970=1176.819,74.634,-49.902,-179.227,6.090,148.866
C00971=1176.813,74.883,-49.919,-179.224,6.092,148.865
C00972=1176.808,75.133,-49.935,-179.222,6.093,148.865
C00973=1176.803,75.383,-49.953,-179.220,6.093,148.864
C00974=1176.799,75.632,-49.969,-179.217,6.095,148.864
C00975=1176.794,75.881,-49.987,-179.214,6.096,148.863
C00976=1176.789,76.130,-50.004,-179.211,6.097,148.862
C00977=1176.783,76.380,-50.021,-179.209,6.098,148.862
C00978=1176.778,76.629,-50.039,-179.206,6.099,148.861
C00979=1176.774,76.878,-50.056,-179.204,6.100,148.861
C00980=1176.769,77.128,-50.073,-179.201,6.101,148.860
C00981=1176.765,77.377,-50.090,-179.198,6.102,148.860
C00982=1176.759,77.627,-50.108,-179.196,6.103,148.859
C00983=1176.754,77.876,-50.124,-179.193,6.105,148.859
C00984=1176.749,78.125,-50.142,-179.190,6.105,148.858
C00985=1176.744,78.375,-50.159,-179.188,6.107,148.858
C00986=1176.740,78.624,-50.176,-179.185,6.107,148.857
C00987=1176.735,78.873,-50.194,-179.182,6.109,148.857
C00988=1176.730,79.123,-50.211,-179.180,6.110,148.856
C00989=1176.725,79.373,-50.228,-179.177,6.111,148.856
C00990=1176.720,79.621,-50.245,-179.174,6.112,148.855
C00991=1176.714,79.871,-50.263,-179.172,6.114,148.854
C00992=1176.710,80.139,-50.281,-179.169,6.114,148.854
C00993=1176.705,80.408,-50.300,-179.166,6.116,148.853
C00994=1176.699,80.676,-50.318,-179.164,6.116,148.853
C00995=1176.693,80.944,-50.338,-179.160,6.118,148.852
C00996=1176.689,81.194,-50.354,-179.158,6.119,148.852
C00997=1176.684,81.443,-50.372,-179.156,6.120,148.851
C00998=1176.679,81.693,-50.390,-179.152,6.122,148.851
C00999=1176.674,81.942,-50.408,-179.150,6.122,148.850
C01000=1176.669,82.191,-50.424,-179.147,6.124,148.850
C01001=1176.665,82.440,-50.442,-179.145,6.125,148.849
C01002=1176.659,82.690,-50.460,-179.142,6.125,148.848
C01003=1176.654,82.939,-50.478,-179.140,6.127,148.848
C01004=1176.649,83.188,-50.494,-179.137,6.127,148.847
C01005=1176.644,83.437,-50.512,-179.134,6.129,148.847
C01006=1176.639,83.687,-50.529,-179.132,6.130,148.846
C01007=1176.634,83.936,-50.547,-179.129,6.131,148.846
C01008=1176.630,84.186,-50.564,-179.127,6.132,148.845
C01009=1176.625,84.435,-50.582,-179.123,6.134,148.845
C01010=1176.620,84.684,-50.600,-179.121,6.135,148.844
C01011=1176.615,84.934,-50.617,-179.118,6.136,148.844
C01012=1176.610,85.183,-50.635,-179.116,6.137,148.843
C01013=1176.606,85.432,-50.652,-179.113,6.138,148.843
C01014=1176.600,85.682,-50.670,-179.111,6.139,148.842
C01015=1176.596,85.931,-50.688,-179.108,6.141,148.842
C01016=1176.590,86.181,-50.705,-179.105,6.141,148.841
C01017=1176.585,86.430,-50.723,-179.103,6.143,148.841
C01018=1176.581,86.679,-50.740,-179.100,6.144,148.840
C01019=1176.576,86.928,-50.758,-179.097,6.145,148.840
C01020=1176.571,87.178,-50.775,-179.095,6.146,148.839
C01021=1176.566,87.427,-50.793,-179.092,6.148,148.839
C01022=1176.561,87.676,-50.811,-179.090,6.148,148.838
C01023=1176.556,87.926,-50.829,-179.087,6.150,148.838
C01024=1176.551,88.175,-50.847,-179.084,6.151,148.837
C01025=1176.546,88.424,-50.865,-179.081,6.152,148.836
C01026=1176.541,88.673,-50.883,-179.079,6.153,148.836
C01027=1176.537,88.923,-50.899,-179.076,6.154,148.835
C01028=1176.532,89.172,-50.917,-179.073,6.156,148.835
C01029=1176.528,89.422,-50.936,-179.071,6.157,148.835
C01030=1176.523,89.671,-50.954,-179.068,6.158,148.834
C01031=1176.518,89.920,-50.972,-179.066,6.159,148.833
C01032=1176.513,90.170,-50.989,-179.062,6.160,148.833
C01033=1176.508,90.419,-51.007,-179.060,6.161,148.832
C01034=1176.503,90.668,-51.025,-179.057,6.163,148.832
C01035=1176.498,90.918,-51.043,-179.055,6.164,148.831
C01036=1176.493,91.167,-51.061,-179.052,6.165,148.831
C01037=1176.488,91.416,-51.079,-179.050,6.166,148.830
C01038=1176.483,91.665,-51.097,-179.047,6.168,148.830
C01039=1176.478,91.915,-51.114,-179.044,6.168,148.829
C01040=1176.473,92.164,-51.132,-179.042,6.170,148.829
C01041=1176.469,92.414,-51.150,-179.039,6.171,148.828
C01042=1176.464,92.663,-51.168,-179.036,6.172,148.828
C01043=1176.459,92.912,-51.186,-179.034,6.174,148.827
C01044=1176.454,93.161,-51.204,-179.031,6.174,148.827
C01045=1176.449,93.411,-51.222,-179.028,6.176,148.826
C01046=1176.444,93.660,-51.240,-179.026,6.177,148.826
C01047=1176.439,93.909,-51.258,-179.023,6.178,148.825
C01048=1176.434,94.158,-51.276,-179.021,6.179,148.825
C01049=1176.430,94.408,-51.295,-179.017,6.181,148.824
C01050=1176.425,94.657,-51.312,-179.015,6.182,148.824
C01051=1176.420,94.906,-51.330,-179.013,6.183,148.823
C01052=1176.415,95.156,-51.348,-179.009,6.185,148.823
C01053=1176.410,95.405,-51.366,-179.007,6.186,148.822
C01054=1176.405,95.654,-51.384,-179.004,6.187,148.822
C01055=1176.400,95.903,-51.403,-179.002,6.188,148.821
C01056=1176.395,96.153,-51.421,-178.999,6.189,148.821
C01057=1176.391,96.402,-51.439,-178.997,6.190,148.820
C01058=1176.386,96.652,-51.457,-178.994,6.192,148.820
C01059=1176.381,96.901,-51.475,-178.991,6.193,148.819
C01060=1176.376,97.150,-51.493,-178.989,6.194,148.819
C01061=1176.372,97.399,-51.512,-178.986,6.196,148.818
C01062=1176.367,97.648,-51.530,-178.983,6.196,148.818
C01063=1176.361,97.898,-51.549,-178.981,6.198,148.817
C01064=1176.356,98.147,-51.567,-178.978,6.199,148.817
C01065=1176.351,98.396,-51.585,-178.975,6.200,148.816
C01066=1176.347,98.646,-51.603,-178.972,6.202,148.816
C01067=1176.342,98.895,-51.621,-178.970,6.203,148.815
C01068=1176.338,99.144,-51.640,-178.967,6.204,148.815
C01069=1176.332,99.393,-51.658,-178.965,6.205,148.814
C01070=1176.328,99.643,-51.677,-178.962,6.207,148.814
C01071=1176.323,99.892,-51.695,-178.959,6.208,148.813
C01072=1176.318,100.142,-51.713,-178.957,6.209,148.813
C01073=1176.313,100.390,-51.731,-178.954,6.210,148.812
C01074=1176.308,100.640,-51.750,-178.952,6.211,148.812
C01075=1176.303,100.890,-51.768,-178.949,6.213,148.811
C01076=1176.298,101.139,-51.786,-178.946,6.214,148.811
C01077=1176.294,101.387,-51.805,-178.944,6.215,148.810
C01078=1176.289,101.637,-51.824,-178.941,6.217,148.810
C01079=1176.284,101.887,-51.842,-178.938,6.218,148.809
C01080=1176.279,102.136,-51.860,-178.936,6.219,148.809
C01081=1176.274,102.384,-51.879,-178.932,6.221,148.808
C01082=1176.269,102.635,-51.898,-178.930,6.222,148.808
C01083=1176.264,102.884,-51.916,-178.927,6.223,148.807
C01084=1176.260,103.132,-51.934,-178.925,6.224,148.807
C01085=1176.255,103.382,-51.953,-178.922,6.226,148.806
C01086=1176.250,103.632,-51.971,-178.919,6.227,148.806
C01087=1176.245,103.880,-51.990,-178.917,6.228,148.805
C01088=1176.239,104.130,-52.008,-178.914,6.230,148.805
C01089=1176.235,104.379,-52.027,-178.912,6.231,148.804
C01090=1176.231,104.628,-52.045,-178.909,6.232,148.804
C01091=1176.225,104.878,-52.064,-178.906,6.234,148.803
C01092=1176.221,105.127,-52.083,-178.904,6.235,148.803
C01093=1176.216,105.376,-52.101,-178.901,6.236,148.802
C01094=1176.211,105.625,-52.120,-178.898,6.238,148.802
C01095=1176.206,105.875,-52.139,-178.896,6.239,148.801
C01096=1176.201,106.143,-52.159,-178.893,6.240,148.801
C01097=1176.196,106.411,-52.179,-178.890,6.242,148.800
C01098=1176.191,106.680,-52.199,-178.887,6.243,148.800
C01099=1176.186,106.948,-52.219,-178.884,6.245,148.799
C01100=1176.180,107.197,-52.238,-178.881,6.245,148.799
C01101=1176.176,107.447,-52.257,-178.879,6.247,148.798
C01102=1176.171,107.696,-52.275,-178.876,6.249,148.798
C01103=1176.166,107.945,-52.294,-178.873,6.249,148.797
C01104=1176.162,108.195,-52.313,-178.871,6.251,148.797
C01105=1176.156,108.443,-52.332,-178.869,6.252,148.796
C01106=1176.152,108.693,-52.350,-178.865,6.253,148.796
C01107=1176.147,108.942,-52.370,-178.863,6.255,148.795
C01108=1176.142,109.191,-52.388,-178.861,6.256,148.795
C01109=1176.137,109.441,-52.407,-178.857,6.257,148.794
C01110=1176.132,109.689,-52.426,-178.855,6.259,148.794
C01111=1176.127,109.940,-52.445,-178.852,6.260,148.794
C01112=1176.123,110.188,-52.463,-178.849,6.261,148.793
C01113=1176.118,110.438,-52.483,-178.847,6.263,148.792
C01114=1176.113,110.687,-52.501,-178.844,6.264,148.792
C01115=1176.108,110.936,-52.520,-178.841,6.265,148.791
C01116=1176.103,111.186,-52.539,-178.839,6.267,148.791
C01117=1176.098,111.435,-52.558,-178.836,6.268,148.791
C01118=1176.094,111.684,-52.577,-178.834,6.270,148.790
C01119=1176.089,111.933,-52.596,-178.830,6.271,148.790
C01120=1176.084,112.183,-52.615,-178.828,6.272,148.789
C01121=1176.079,112.431,-52.634,-178.826,6.274,148.789
C01122=1176.075,112.681,-52.653,-178.822,6.275,148.788
C01123=1176.069,112.930,-52.672,-178.820,6.276,148.788
C01124=1176.065,113.180,-52.691,-178.818,6.278,148.787
C01125=1176.060,113.428,-52.710,-178.814,6.279,148.787
C01126=1176.055,113.678,-52.730,-178.812,6.281,148.786
C01127=1176.050,113.927,-52.748,-178.810,6.282,148.786
C01128=1176.045,114.176,-52.767,-178.807,6.283,148.785
C01129=1176.040,114.425,-52.787,-178.804,6.285,148.785
C01130=1176.036,114.674,-52.805,-178.802,6.286,148.784
C01131=1176.031,114.924,-52.825,-178.799,6.287,148.784
C01132=1176.026,115.173,-52.843,-178.796,6.289,148.783
C01133=1176.021,115.422,-52.863,-178.794,6.290,148.783
C01134=1176.016,115.672,-52.882,-178.791,6.292,148.783
C01135=1176.012,115.920,-52.901,-178.788,6.293,148.782
C01136=1176.007,116.170,-52.921,-178.786,6.294,148.782
C01137=1176.002,116.419,-52.940,-178.783,6.296,148.781
C01138=1175.998,116.668,-52.959,-178.780,6.297,148.781
C01139=1175.992,116.918,-52.978,-178.777,6.299,148.780
C01140=1175.987,117.167,-52.997,-178.775,6.300,148.780
C01141=1175.982,117.416,-53.016,-178.772,6.301,148.779
C01142=1175.978,117.665,-53.036,-178.769,6.303,148.779
C01143=1175.973,117.914,-53.055,-178.767,6.304,148.778
C01144=1175.968,118.164,-53.074,-178.764,6.305,148.778
C01145=1175.964,118.413,-53.094,-178.761,6.307,148.777
C01146=1175.959,118.662,-53.113,-178.759,6.309,148.777
C01147=1175.954,118.911,-53.132,-178.756,6.309,148.776
C01148=1175.949,119.160,-53.152,-178.753,6.311,148.776
C01149=1175.945,119.410,-53.171,-178.751,6.313,148.776
C01150=1175.939,119.658,-53.190,-178.748,6.314,148.775
C01151=1175.934,119.908,-53.210,-178.745,6.315,148.775
C01152=1175.930,120.158,-53.229,-178.743,6.317,148.774
C01153=1175.925,120.406,-53.248,-178.740,6.319,148.774
C01154=1175.920,120.656,-53.268,-178.738,6.319,148.773
C01155=1175.916,120.905,-53.287,-178.735,6.321,148.773
C01156=1175.910,121.154,-53.307,-178.732,6.323,148.772
C01157=1175.905,121.404,-53.326,-178.729,6.324,148.772
C01158=1175.901,121.652,-53.346,-178.727,6.325,148.772
C01159=1175.896,121.901,-53.365,-178.724,6.327,148.771
C01160=1175.892,122.151,-53.385,-178.721,6.328,148.771
C01161=1175.886,122.400,-53.404,-178.718,6.330,148.770
C01162=1175.882,122.649,-53.424,-178.716,6.331,148.770
C01163=1175.877,122.899,-53.444,-178.713,6.332,148.769
C01164=1175.872,123.147,-53.462,-178.710,6.334,148.769
C01165=1175.868,123.397,-53.482,-178.708,6.336,148.768
C01166=1175.863,123.646,-53.502,-178.706,6.337,148.768
C01167=1175.858,123.895,-53.522,-178.702,6.338,148.767
C01168=1175.853,124.144,-53.541,-178.700,6.340,148.767
C01169=1175.848,124.394,-53.561,-178.697,6.342,148.767
C01170=1175.843,124.643,-53.580,-178.695,6.343,148.766
C01171=1175.838,124.892,-53.601,-178.692,6.344,148.765
C01172=1175.834,125.141,-53.620,-178.689,6.346,148.765
C01173=1175.829,125.390,-53.639,-178.686,6.347,148.765
C01174=1175.824,125.639,-53.659,-178.684,6.348,148.764
C01175=1175.820,125.888,-53.679,-178.681,6.350,148.764
C01176=1175.815,126.138,-53.699,-178.678,6.351,148.763
C01177=1175.810,126.387,-53.718,-178.676,6.353,148.763
C01178=1175.805,126.636,-53.738,-178.673,6.354,148.762
C01179=1175.801,126.885,-53.758,-178.671,6.356,148.762
C01180=1175.796,127.135,-53.778,-178.668,6.357,148.761
C01181=1175.791,127.383,-53.798,-178.665,6.359,148.761
C01182=1175.786,127.633,-53.817,-178.662,6.361,148.761
C01183=1175.781,127.882,-53.837,-178.660,6.362,148.760
C01184=1175.777,128.131,-53.857,-178.657,6.363,148.760
C01185=1175.772,128.380,-53.877,-178.654,6.365,148.759
C01186=1175.767,128.630,-53.896,-178.651,6.367,148.759
C01187=1175.762,128.879,-53.917,-178.649,6.367,148.758
C01188=1175.758,129.128,-53.936,-178.647,6.369,148.758
C01189=1175.753,129.376,-53.956,-178.644,6.371,148.758
C01190=1175.748,129.626,-53.976,-178.641,6.372,148.757
C01191=1175.744,129.875,-53.996,-178.638,6.374,148.757
C01192=1175.739,130.124,-54.016,-178.636,6.375,148.756
C01193=1175.733,130.373,-54.035,-178.633,6.377,148.756
C01194=1175.729,130.622,-54.056,-178.630,6.378,148.755
C01195=1175.723,130.872,-54.076,-178.627,6.380,148.755
C01196=1175.719,131.121,-54.096,-178.625,6.382,148.754
C01197=1175.714,131.371,-54.116,-178.622,6.383,148.754
C01198=1175.709,131.619,-54.136,-178.620,6.384,148.754
C01199=1175.705,131.869,-54.156,-178.617,6.386,148.753
C01200=1175.700,132.137,-54.177,-178.614,6.387,148.753
C01201=1175.694,132.405,-54.199,-178.611,6.389,148.752
C01202=1175.689,132.674,-54.220,-178.608,6.391,148.752
C01203=1175.684,132.942,-54.243,-178.605,6.392,148.751
C01204=1175.679,133.192,-54.262,-178.603,6.394,148.751
C01205=1175.675,133.441,-54.283,-178.600,6.396,148.750
C01206=1175.670,133.690,-54.303,-178.597,6.397,148.750
C01207=1175.666,133.940,-54.323,-178.595,6.398,148.749
C01208=1175.660,134.189,-54.344,-178.592,6.400,148.749
C01209=1175.655,134.438,-54.363,-178.589,6.402,148.749
C01210=1175.651,134.687,-54.383,-178.586,6.403,148.748
C01211=1175.646,134.936,-54.404,-178.584,6.405,148.748
C01212=1175.642,135.185,-54.423,-178.581,6.407,148.748
C01213=1175.636,135.434,-54.444,-178.578,6.407,148.747
C01214=1175.632,135.683,-54.465,-178.576,6.409,148.746
C01215=1175.627,135.933,-54.484,-178.573,6.411,148.746
C01216=1175.623,136.182,-54.505,-178.570,6.413,148.746
C01217=1175.618,136.431,-54.526,-178.568,6.414,148.745
C01218=1175.613,136.679,-54.546,-178.565,6.416,148.745
C01219=1175.608,136.929,-54.565,-178.563,6.417,148.745
C01220=1175.603,137.178,-54.586,-178.560,6.418,148.744
C01221=1175.598,137.427,-54.607,-178.557,6.420,148.744
C01222=1175.594,137.676,-54.627,-178.554,6.422,148.743
C01223=1175.589,137.926,-54.647,-178.552,6.424,148.743
C01224=1175.585,138.175,-54.667,-178.549,6.425,148.742
C01225=1175.579,138.424,-54.688,-178.546,6.427,148.742
C01226=1175.575,138.673,-54.708,-178.544,6.428,148.741
C01227=1175.570,138.922,-54.729,-178.541,6.429,148.741
C01228=1175.565,139.171,-54.750,-178.538,6.431,148.741
C01229=1175.561,139.421,-54.769,-178.535,6.433,148.740
C01230=1175.556,139.670,-54.790,-178.533,6.435,148.740
C01231=1175.551,139.919,-54.811,-178.530,6.436,148.739
C01232=1175.547,140.168,-54.831,-178.527,6.438,148.739
C01233=1175.542,140.417,-54.852,-178.525,6.439,148.739
C01234=1175.537,140.666,-54.872,-178.522,6.441,148.738
C01235=1175.532,140.915,-54.893,-178.519,6.442,148.738
C01236=1175.528,141.164,-54.913,-178.517,6.444,148.737
C01237=1175.523,141.413,-54.934,-178.514,6.446,148.737
C01238=1175.518,141.663,-54.954,-178.511,6.448,148.736
C01239=1175.513,141.912,-54.975,-178.509,6.449,148.736
C01240=1175.509,142.161,-54.995,-178.506,6.451,148.736
C01241=1175.504,142.410,-55.016,-178.503,6.452,148.735
C01242=1175.499,142.659,-55.037,-178.501,6.453,148.735
C01243=1175.494,142.908,-55.057,-178.498,6.455,148.734
C01244=1175.489,143.157,-55.078,-178.495,6.457,148.734
C01245=1175.485,143.406,-55.098,-178.493,6.459,148.734
C01246=1175.480,143.656,-55.119,-178.490,6.460,148.733
C01247=1175.475,143.904,-55.140,-178.487,6.462,148.733
C01248=1175.470,144.154,-55.161,-178.484,6.464,148.732
C01249=1175.466,144.402,-55.182,-178.482,6.466,148.732
C01250=1175.461,144.651,-55.202,-178.479,6.466,148.731
C01251=1175.456,144.900,-55.223,-178.476,6.468,148.731
C01252=1175.452,145.149,-55.243,-178.474,6.470,148.731
C01253=1175.447,145.398,-55.264,-178.471,6.471,148.730
C01254=1175.442,145.647,-55.285,-178.468,6.473,148.730
C01255=1175.437,145.897,-55.306,-178.466,6.475,148.729
C01256=1175.433,146.146,-55.326,-178.463,6.477,148.729
C01257=1175.428,146.396,-55.347,-178.460,6.478,148.729
C01258=1175.423,146.644,-55.369,-178.458,6.480,148.728
C01259=1175.419,146.893,-55.389,-178.455,6.482,148.728
C01260=1175.414,147.142,-55.410,-178.452,6.484,148.728
C01261=1175.409,147.391,-55.431,-178.450,6.484,148.727
C01262=1175.404,147.641,-55.452,-178.447,6.486,148.727
C01263=1175.400,147.889,-55.473,-178.444,6.488,148.726
C01264=1175.395,148.138,-55.494,-178.442,6.490,148.726
C01265=1175.390,148.388,-55.515,-178.439,6.491,148.725
C01266=1175.386,148.637,-55.535,-178.436,6.493,148.725
C01267=1175.380,148.886,-55.556,-178.433,6.495,148.725
C01268=1175.376,149.135,-55.578,-178.431,6.497,148.724
C01269=1175.371,149.384,-55.598,-178.428,6.498,148.724
C01270=1175.366,149.633,-55.619,-178.425,6.500,148.724
C01271=1175.362,149.882,-55.641,-178.423,6.502,148.723
C01272=1175.357,150.132,-55.662,-178.420,6.504,148.723
C01273=1175.352,150.381,-55.683,-178.417,6.505,148.722
C01274=1175.348,150.629,-55.704,-178.414,6.507,148.722
C01275=1175.343,150.878,-55.725,-178.412,6.508,148.721
C01276=1175.338,151.128,-55.746,-178.409,6.509,148.721
C01277=1175.334,151.376,-55.767,-178.407,6.511,148.721
C01278=1175.329,151.626,-55.788,-178.404,6.513,148.720
C01279=1175.324,151.875,-55.809,-178.401,6.515,148.720
C01280=1175.320,152.124,-55.830,-178.399,6.516,148.719
C01281=1175.314,152.373,-55.851,-178.396,6.518,148.719
C01282=1175.310,152.621,-55.873,-178.393,6.520,148.719
C01283=1175.305,152.871,-55.894,-178.390,6.522,148.718
C01284=1175.301,153.120,-55.915,-178.388,6.523,148.718
C01285=1175.296,153.369,-55.936,-178.385,6.525,148.718
C01286=1175.291,153.618,-55.957,-178.382,6.527,148.717
C01287=1175.286,153.867,-55.979,-178.380,6.529,148.717
C01288=1175.282,154.117,-56.000,-178.377,6.530,148.716
C01289=1175.277,154.365,-56.021,-178.374,6.532,148.716
C01290=1175.272,154.614,-56.042,-178.372,6.534,148.716
C01291=1175.267,154.863,-56.064,-178.369,6.536,148.715
C01292=1175.263,155.113,-56.085,-178.366,6.537,148.715
C01293=1175.258,155.361,-56.107,-178.364,6.539,148.715
C01294=1175.253,155.611,-56.127,-178.360,6.541,148.714
C01295=1175.248,155.859,-56.149,-178.358,6.542,148.714
C01296=1175.244,156.109,-56.171,-178.355,6.544,148.713
C01297=1175.239,156.358,-56.192,-178.352,6.546,148.713
C01298=1175.235,156.606,-56.213,-178.350,6.548,148.712
C01299=1175.230,156.856,-56.235,-178.347,6.549,148.712
C01300=1175.225,157.105,-56.256,-178.344,6.551,148.712
C01301=1175.220,157.353,-56.278,-178.342,6.553,148.711
C01302=1175.215,157.603,-56.299,-178.339,6.555,148.711
C01303=1175.211,157.852,-56.321,-178.336,6.556,148.711
C01304=1175.206,158.121,-56.344,-178.334,6.558,148.710
C01305=1175.201,158.390,-56.367,-178.331,6.560,148.710
C01306=1175.196,158.659,-56.391,-178.328,6.562,148.709
C01307=1175.190,158.928,-56.414,-178.325,6.564,148.709
C01308=1175.186,159.177,-56.436,-178.323,6.565,148.709
C01309=1175.181,159.426,-56.456,-178.320,6.567,148.708
C01310=1175.177,159.674,-56.478,-178.317,6.569,148.708
C01311=1175.172,159.924,-56.500,-178.315,6.571,148.708
C01312=1175.167,160.172,-56.521,-178.312,6.572,148.707
C01313=1175.163,160.422,-56.543,-178.309,6.574,148.707
C01314=1175.158,160.671,-56.564,-178.307,6.576,148.706
C01315=1175.153,160.920,-56.586,-178.304,6.578,148.706
C01316=1175.149,161.169,-56.608,-178.301,6.580,148.706
C01317=1175.144,161.418,-56.630,-178.298,6.582,148.705
C01318=1175.139,161.667,-56.651,-178.295,6.584,148.705
C01319=1175.134,161.916,-56.673,-178.293,6.585,148.705
C01320=1175.130,162.165,-56.695,-178.290,6.587,148.704
C01321=1175.125,162.414,-56.717,-178.287,6.589,148.704
C01322=1175.120,162.663,-56.738,-178.285,6.591,148.704
C01323=1175.116,162.912,-56.760,-178.282,6.592,148.703
C01324=1175.111,163.161,-56.782,-178.279,6.594,148.703
C01325=1175.106,163.409,-56.804,-178.277,6.596,148.702
C01326=1175.102,163.659,-56.825,-178.274,6.598,148.702
C01327=1175.097,163.908,-56.847,-178.271,6.600,148.702
C01328=1175.092,164.157,-56.868,-178.268,6.601,148.701
C01329=1175.088,164.406,-56.890,-178.266,6.603,148.701
C01330=1175.083,164.655,-56.912,-178.263,6.605,148.701
C01331=1175.079,164.904,-56.934,-178.260,6.607,148.700
C01332=1175.073,165.153,-56.956,-178.258,6.608,148.700
C01333=1175.069,165.402,-56.978,-178.255,6.610,148.699
C01334=1175.064,165.651,-57.000,-178.252,6.612,148.699
C01335=1175.060,165.900,-57.022,-178.250,6.614,148.699
C01336=1175.055,166.149,-57.044,-178.247,6.615,148.698
C01337=1175.051,166.398,-57.066,-178.244,6.617,148.698
C01338=1175.046,166.647,-57.088,-178.242,6.619,148.698
C01339=1175.041,166.896,-57.110,-178.239,6.621,148.697
C01340=1175.036,167.145,-57.132,-178.236,6.622,148.697
C01341=1175.032,167.395,-57.154,-178.234,6.624,148.696
C01342=1175.027,167.643,-57.176,-178.231,6.626,148.696
C01343=1175.022,167.891,-57.198,-178.228,6.629,148.696
C01344=1175.018,168.141,-57.220,-178.225,6.630,148.695
C01345=1175.013,168.389,-57.242,-178.223,6.632,148.695
C01346=1175.008,168.639,-57.264,-178.220,6.634,148.695
C01347=1175.004,168.888,-57.287,-178.217,6.636,148.695
C01348=1174.999,169.137,-57.308,-178.215,6.638,148.694
C01349=1174.995,169.386,-57.330,-178.212,6.640,148.694
C01350=1174.989,169.635,-57.353,-178.209,6.641,148.693
C01351=1174.985,169.884,-57.375,-178.207,6.643,148.693
C01352=1174.980,170.133,-57.397,-178.204,6.645,148.693
C01353=1174.976,170.382,-57.419,-178.201,6.647,148.692
C01354=1174.970,170.631,-57.441,-178.199,6.648,148.692
C01355=1174.966,170.880,-57.464,-178.196,6.650,148.692
C01356=1174.961,171.128,-57.486,-178.193,6.652,148.691
C01357=1174.957,171.378,-57.508,-178.190,6.654,148.691
C01358=1174.952,171.626,-57.530,-178.187,6.656,148.691
C01359=1174.948,171.875,-57.553,-178.185,6.658,148.690
C01360=1174.943,172.125,-57.575,-178.182,6.660,148.690
C01361=1174.938,172.373,-57.597,-178.180,6.662,148.690
C01362=1174.934,172.622,-57.620,-178.177,6.664,148.689
C01363=1174.929,172.871,-57.642,-178.174,6.665,148.689
C01364=1174.924,173.120,-57.664,-178.172,6.667,148.689
C01365=1174.920,173.369,-57.687,-178.169,6.669,148.688
C01366=1174.915,173.618,-57.709,-178.166,6.671,148.688
C01367=1174.910,173.868,-57.731,-178.164,6.672,148.687
C01368=1174.906,174.116,-57.754,-178.160,6.675,148.687
C01369=1174.901,174.365,-57.776,-178.158,6.677,148.687
C01370=1174.896,174.615,-57.798,-178.155,6.679,148.687
C01371=1174.892,174.863,-57.821,-178.153,6.681,148.686
C01372=1174.887,175.112,-57.843,-178.150,6.682,148.686
C01373=1174.883,175.361,-57.866,-178.147,6.684,148.686
C01374=1174.878,175.610,-57.888,-178.145,6.686,148.685
C01375=1174.873,175.859,-57.911,-178.142,6.688,148.685
C01376=1174.869,176.108,-57.933,-178.139,6.690,148.684
C01377=1174.864,176.356,-57.956,-178.136,6.692,148.684
C01378=1174.859,176.606,-57.978,-178.133,6.694,148.684
C01379=1174.855,176.855,-58.002,-178.131,6.696,148.684
C01380=1174.850,177.103,-58.023,-178.129,6.698,148.683
C01381=1174.846,177.352,-58.046,-178.126,6.700,148.683
C01382=1174.841,177.602,-58.069,-178.123,6.701,148.682
C01383=1174.836,177.850,-58.091,-178.121,6.703,148.682
C01384=1174.831,178.099,-58.114,-178.118,6.705,148.682
C01385=1174.827,178.348,-58.137,-178.115,6.707,148.681
C01386=1174.822,178.597,-58.159,-178.112,6.709,148.681
C01387=1174.818,178.846,-58.182,-178.110,6.711,148.681
C01388=1174.813,179.095,-58.205,-178.107,6.713,148.681
C01389=1174.809,179.344,-58.227,-178.104,6.715,148.680
C01390=1174.803,179.592,-58.250,-178.102,6.717,148.680
C01391=1174.799,179.841,-58.273,-178.099,6.718,148.679
C01392=1174.794,180.091,-58.295,-178.096,6.721,148.679
C01393=1174.790,180.340,-58.319,-178.093,6.723,148.679
C01394=1174.785,180.588,-58.341,-178.091,6.725,148.679
C01395=1174.780,180.837,-58.364,-178.088,6.727,148.678
C01396=1174.776,181.086,-58.387,-178.086,6.728,148.678
C01397=1174.772,181.335,-58.410,-178.083,6.730,148.678
C01398=1174.767,181.584,-58.432,-178.080,6.733,148.677
C01399=1174.762,181.833,-58.455,-178.077,6.735,148.677
C01400=1174.757,182.082,-58.478,-178.075,6.737,148.677
C01401=1174.753,182.331,-58.501,-178.072,6.739,148.676
C01402=1174.748,182.580,-58.523,-178.069,6.740,148.676
C01403=1174.744,182.828,-58.546,-178.067,6.742,148.676
C01404=1174.739,183.077,-58.570,-178.063,6.745,148.675
C01405=1174.734,183.326,-58.593,-178.061,6.746,148.675
C01406=1174.730,183.575,-58.616,-178.058,6.748,148.675
C01407=1174.725,183.824,-58.638,-178.056,6.750,148.674
C01408=1174.719,184.094,-58.663,-178.053,6.752,148.674
C01409=1174.715,184.363,-58.688,-178.050,6.755,148.674
C01410=1174.710,184.632,-58.713,-178.047,6.756,148.673
C01411=1174.705,184.903,-58.739,-178.044,6.759,148.673
C01412=1174.701,185.151,-58.761,-178.041,6.761,148.673
C01413=1174.696,185.400,-58.784,-178.039,6.763,148.672
C01414=1174.691,185.649,-58.808,-178.036,6.764,148.672
C01415=1174.686,185.899,-58.830,-178.033,6.767,148.672
C01416=1174.682,186.147,-58.853,-178.031,6.769,148.672
C01417=1174.677,186.396,-58.876,-178.028,6.771,148.671
C01418=1174.672,186.645,-58.899,-178.025,6.773,148.671
C01419=1174.668,186.893,-58.922,-178.023,6.774,148.670
C01420=1174.664,187.142,-58.946,-178.020,6.776,148.670
C01421=1174.659,187.392,-58.969,-178.017,6.779,148.670
C01422=1174.654,187.641,-58.992,-178.014,6.781,148.670
C01423=1174.649,187.890,-59.016,-178.012,6.783,148.669
C01424=1174.645,188.138,-59.038,-178.009,6.784,148.669
C01425=1174.641,188.387,-59.062,-178.006,6.787,148.669
C01426=1174.636,188.636,-59.085,-178.004,6.789,148.668
C01427=1174.631,188.885,-59.108,-178.001,6.791,148.668
C01428=1174.626,189.134,-59.131,-177.998,6.793,148.668
C01429=1174.622,189.382,-59.156,-177.996,6.795,148.667
C01430=1174.618,189.631,-59.178,-177.993,6.797,148.667
C01431=1174.613,189.880,-59.202,-177.990,6.799,148.667
C01432=1174.608,190.129,-59.225,-177.987,6.801,148.667
C01433=1174.604,190.378,-59.248,-177.985,6.803,148.666
C01434=1174.599,190.627,-59.272,-177.982,6.805,148.666
C01435=1174.594,190.876,-59.295,-177.979,6.808,148.666
C01436=1174.589,191.125,-59.318,-177.977,6.809,148.665
C01437=1174.585,191.373,-59.343,-177.974,6.811,148.665
C01438=1174.581,191.622,-59.365,-177.971,6.813,148.665
C01439=1174.576,191.871,-59.389,-177.969,6.816,148.665
C01440=1174.572,192.120,-59.412,-177.966,6.818,148.664
C01441=1174.567,192.369,-59.435,-177.963,6.819,148.664
C01442=1174.563,192.618,-59.459,-177.961,6.821,148.664
C01443=1174.558,192.867,-59.483,-177.958,6.823,148.663
C01444=1174.553,193.115,-59.506,-177.955,6.826,148.663
C01445=1174.548,193.364,-59.529,-177.952,6.828,148.663
C01446=1174.544,193.612,-59.553,-177.950,6.829,148.662
C01447=1174.539,193.862,-59.577,-177.948,6.832,148.662
C01448=1174.534,194.111,-59.600,-177.944,6.834,148.662
C01449=1174.530,194.359,-59.624,-177.942,6.836,148.662
C01450=1174.526,194.609,-59.648,-177.939,6.838,148.661
C01451=1174.521,194.858,-59.671,-177.937,6.840,148.661
C01452=1174.517,195.106,-59.695,-177.934,6.842,148.661
C01453=1174.512,195.355,-59.719,-177.931,6.844,148.660
C01454=1174.507,195.604,-59.742,-177.928,6.846,148.660
C01455=1174.503,195.853,-59.766,-177.926,6.848,148.660
C01456=1174.498,196.102,-59.789,-177.923,6.851,148.660
C01457=1174.494,196.350,-59.813,-177.920,6.853,148.659
C01458=1174.489,196.599,-59.837,-177.917,6.854,148.659
C01459=1174.484,196.848,-59.860,-177.915,6.857,148.659
C01460=1174.480,197.097,-59.884,-177.912,6.859,148.658
C01461=1174.474,197.346,-59.908,-177.909,6.861,148.658
C01462=1174.470,197.594,-59.932,-177.907,6.863,148.658
C01463=1174.465,197.843,-59.956,-177.904,6.866,148.658
C01464=1174.461,198.092,-59.980,-177.901,6.867,148.657
C01465=1174.456,198.341,-60.003,-177.899,6.869,148.657
C01466=1174.452,198.589,-60.027,-177.896,6.871,148.657
C01467=1174.448,198.839,-60.051,-177.893,6.874,148.657
C01468=1174.443,199.087,-60.075,-177.890,6.876,148.656
C01469=1174.439,199.336,-60.098,-177.888,6.877,148.656
C01470=1174.434,199.585,-60.123,-177.885,6.880,148.656
C01471=1174.429,199.834,-60.147,-177.882,6.882,148.655
C01472=1174.424,200.083,-60.170,-177.880,6.884,148.655
C01473=1174.420,200.331,-60.194,-177.877,6.886,148.655
C01474=1174.415,200.580,-60.218,-177.874,6.889,148.655
C01475=1174.412,200.829,-60.242,-177.872,6.890,148.654
C01476=1174.406,201.078,-60.267,-177.869,6.893,148.654
C01477=1174.402,201.327,-60.290,-177.866,6.895,148.654
C01478=1174.397,201.575,-60.314,-177.863,6.897,148.653
C01479=1174.393,201.824,-60.338,-177.861,6.899,148.653
C01480=1174.388,202.073,-60.362,-177.858,6.902,148.653
C01481=1174.384,202.322,-60.387,-177.855,6.903,148.653
C01482=1174.379,202.571,-60.411,-177.853,6.905,148.652
C01483=1174.375,202.820,-60.434,-177.850,6.907,148.652
C01484=1174.369,203.068,-60.459,-177.847,6.910,148.652
C01485=1174.365,203.317,-60.483,-177.845,6.912,148.652
C01486=1174.361,203.565,-60.507,-177.842,6.914,148.651
C01487=1174.357,203.815,-60.531,-177.839,6.916,148.651
C01488=1174.351,204.064,-60.555,-177.836,6.918,148.651
C01489=1174.347,204.312,-60.580,-177.834,6.920,148.651
C01490=1174.343,204.560,-60.604,-177.831,6.923,148.650
C01491=1174.338,204.810,-60.628,-177.828,6.925,148.650
C01492=1174.333,205.059,-60.652,-177.826,6.927,148.650
C01493=1174.329,205.307,-60.676,-177.823,6.930,148.650
C01494=1174.324,205.556,-60.701,-177.820,6.931,148.649
C01495=1174.320,205.804,-60.725,-177.818,6.933,148.649
C01496=1174.316,206.054,-60.749,-177.815,6.936,148.649
C01497=1174.311,206.302,-60.774,-177.812,6.938,148.648
C01498=1174.306,206.551,-60.797,-177.810,6.940,148.648
C01499=1174.301,206.800,-60.822,-177.807,6.943,148.648
C01500=1174.297,207.049,-60.846,-177.805,6.945,148.648
C01501=1174.293,207.298,-60.870,-177.802,6.946,148.647
C01502=1174.287,207.546,-60.895,-177.799,6.949,148.647
C01503=1174.284,207.795,-60.920,-177.796,6.951,148.647
C01504=1174.279,208.044,-60.944,-177.794,6.953,148.647
C01505=1174.274,208.293,-60.968,-177.791,6.956,148.646
C01506=1174.270,208.541,-60.992,-177.788,6.958,148.646
C01507=1174.265,208.790,-61.017,-177.786,6.960,148.646
C01508=1174.261,209.039,-61.042,-177.782,6.962,148.646
C01509=1174.256,209.287,-61.066,-177.780,6.964,148.645
C01510=1174.252,209.537,-61.091,-177.778,6.966,148.645
C01511=1174.247,209.785,-61.115,-177.775,6.969,148.645
C01512=1174.242,210.056,-61.142,-177.772,6.971,148.645
C01513=1174.237,210.326,-61.169,-177.769,6.973,148.644
C01514=1174.232,210.597,-61.196,-177.766,6.976,148.644
C01515=1174.227,210.867,-61.223,-177.763,6.978,148.644
C01516=1174.223,211.116,-61.247,-177.760,6.981,148.644
C01517=1174.218,211.365,-61.272,-177.758,6.983,148.643
C01518=1174.213,211.613,-61.296,-177.755,6.985,148.643
C01519=1174.209,211.862,-61.321,-177.752,6.987,148.643
C01520=1174.205,212.111,-61.345,-177.749,6.989,148.643
C01521=1174.199,212.360,-61.369,-177.747,6.992,148.642
C01522=1174.196,212.608,-61.395,-177.744,6.994,148.642
C01523=1174.191,212.857,-61.419,-177.742,6.996,148.642
C01524=1174.186,213.105,-61.444,-177.739,6.999,148.642
C01525=1174.182,213.355,-61.468,-177.736,7.000,148.641
C01526=1174.177,213.603,-61.493,-177.734,7.002,148.641
C01527=1174.173,213.852,-61.518,-177.731,7.005,148.641
C01528=1174.168,214.101,-61.543,-177.728,7.007,148.641
C01529=1174.163,214.349,-61.568,-177.725,7.010,148.641
C01530=1174.159,214.598,-61.593,-177.722,7.012,148.640
C01531=1174.154,214.846,-61.617,-177.720,7.014,148.640
C01532=1174.150,215.096,-61.642,-177.717,7.016,148.640
C01533=1174.145,215.344,-61.666,-177.715,7.019,148.640
C01534=1174.141,215.593,-61.692,-177.712,7.021,148.639
C01535=1174.137,215.842,-61.716,-177.709,7.023,148.639
C01536=1174.132,216.090,-61.741,-177.707,7.025,148.639
C01537=1174.127,216.339,-61.767,-177.704,7.028,148.639
C01538=1174.122,216.588,-61.791,-177.701,7.030,148.638
C01539=1174.119,216.836,-61.817,-177.698,7.032,148.638
C01540=1174.114,217.085,-61.841,-177.696,7.035,148.638
C01541=1174.109,217.334,-61.866,-177.693,7.036,148.638
C01542=1174.105,217.582,-61.891,-177.691,7.039,148.638
C01543=1174.101,217.832,-61.916,-177.688,7.041,148.637
C01544=1174.096,218.080,-61.941,-177.685,7.044,148.637
C01545=1174.091,218.329,-61.967,-177.682,7.046,148.637
C01546=1174.087,218.577,-61.991,-177.679,7.048,148.637
C01547=1174.083,218.826,-62.016,-177.677,7.051,148.636
C01548=1174.078,219.074,-62.042,-177.674,7.052,148.636
C01549=1174.073,219.324,-62.067,-177.672,7.055,148.636
C01550=1174.068,219.572,-62.092,-177.669,7.057,148.636
C01551=1174.065,219.821,-62.117,-177.666,7.060,148.636
C01552=1174.060,220.069,-62.142,-177.664,7.062,148.635
C01553=1174.055,220.319,-62.167,-177.661,7.065,148.635
C01554=1174.050,220.567,-62.192,-177.658,7.067,148.635
C01555=1174.046,220.816,-62.218,-177.656,7.069,148.635
C01556=1174.042,221.065,-62.243,-177.653,7.071,148.634
C01557=1174.038,221.313,-62.268,-177.650,7.073,148.634
C01558=1174.033,221.562,-62.293,-177.647,7.076,148.634
C01559=1174.028,221.810,-62.318,-177.645,7.078,148.634
C01560=1174.024,222.059,-62.344,-177.642,7.081,148.634
C01561=1174.019,222.308,-62.369,-177.639,7.083,148.633
C01562=1174.015,222.557,-62.395,-177.637,7.085,148.633
C01563=1174.010,222.805,-62.420,-177.634,7.087,148.633
C01564=1174.006,223.054,-62.444,-177.632,7.090,148.633
C01565=1174.002,223.303,-62.470,-177.628,7.092,148.632
C01566=1173.997,223.551,-62.496,-177.626,7.094,148.632
C01567=1173.992,223.800,-62.521,-177.623,7.097,148.632
C01568=1173.988,224.048,-62.546,-177.621,7.099,148.632
C01569=1173.983,224.297,-62.572,-177.618,7.102,148.632
C01570=1173.979,224.546,-62.597,-177.615,7.104,148.631
C01571=1173.974,224.795,-62.622,-177.612,7.106,148.631
C01572=1173.970,225.043,-62.648,-177.610,7.109,148.631
C01573=1173.965,225.292,-62.673,-177.607,7.111,148.631
C01574=1173.961,225.540,-62.699,-177.604,7.113,148.631
C01575=1173.957,225.789,-62.725,-177.602,7.115,148.630
C01576=1173.952,226.037,-62.750,-177.599,7.118,148.630
C01577=1173.947,226.287,-62.775,-177.596,7.120,148.630
C01578=1173.943,226.535,-62.801,-177.594,7.123,148.630
C01579=1173.938,226.784,-62.826,-177.591,7.125,148.629
C01580=1173.934,227.032,-62.852,-177.588,7.128,148.629
C01581=1173.930,227.281,-62.878,-177.586,7.129,148.629
C01582=1173.925,227.529,-62.903,-177.583,7.132,148.629
C01583=1173.921,227.778,-62.929,-177.581,7.134,148.629
C01584=1173.916,228.027,-62.955,-177.577,7.137,148.629
C01585=1173.912,228.275,-62.980,-177.575,7.139,148.628
C01586=1173.907,228.524,-63.006,-177.572,7.142,148.628
C01587=1173.902,228.773,-63.032,-177.570,7.144,148.628
C01588=1173.898,229.022,-63.058,-177.567,7.147,148.628
C01589=1173.893,229.270,-63.083,-177.564,7.149,148.628
C01590=1173.889,229.519,-63.109,-177.561,7.151,148.627
C01591=1173.885,229.767,-63.135,-177.559,7.153,148.627
C01592=1173.880,230.016,-63.160,-177.556,7.156,148.627
C01593=1173.876,230.264,-63.186,-177.554,7.158,148.627
C01594=1173.872,230.513,-63.212,-177.551,7.161,148.627
C01595=1173.867,230.762,-63.238,-177.548,7.163,148.626
C01596=1173.862,231.010,-63.263,-177.545,7.166,148.626
C01597=1173.858,231.259,-63.289,-177.543,7.168,148.626
C01598=1173.853,231.508,-63.315,-177.540,7.171,148.626
C01599=1173.849,231.757,-63.341,-177.537,7.173,148.626
C01600=1173.844,232.005,-63.366,-177.535,7.175,148.626
C01601=1173.840,232.253,-63.393,-177.532,7.178,148.625
C01602=1173.835,232.502,-63.419,-177.529,7.180,148.625
C01603=1173.831,232.751,-63.445,-177.527,7.182,148.625
C01604=1173.826,232.999,-63.470,-177.524,7.185,148.625
C01605=1173.821,233.248,-63.496,-177.521,7.188,148.625
C01606=1173.817,233.497,-63.522,-177.519,7.190,148.625
C01607=1173.813,233.745,-63.549,-177.516,7.193,148.624
C01608=1173.809,233.994,-63.574,-177.513,7.195,148.624
C01609=1173.803,234.242,-63.600,-177.510,7.197,148.624
C01610=1173.799,234.491,-63.626,-177.508,7.200,148.624
C01611=1173.795,234.739,-63.653,-177.505,7.203,148.624
C01612=1173.790,234.989,-63.679,-177.503,7.204,148.623
C01613=1173.786,235.237,-63.705,-177.500,7.207,148.623
C01614=1173.782,235.486,-63.731,-177.497,7.209,148.623
C01615=1173.777,235.734,-63.756,-177.494,7.212,148.623
C01616=1173.772,236.006,-63.785,-177.491,7.215,148.623
C01617=1173.768,236.277,-63.814,-177.488,7.218,148.623
C01618=1173.763,236.549,-63.842,-177.485,7.220,148.622
C01619=1173.758,236.821,-63.871,-177.483,7.222,148.622
C01620=1173.754,237.069,-63.897,-177.480,7.225,148.622
C01621=1173.749,237.318,-63.924,-177.477,7.228,148.622
C01622=1173.745,237.567,-63.950,-177.475,7.230,148.622
C01623=1173.740,237.814,-63.976,-177.472,7.233,148.622
C01624=1173.735,238.063,-64.002,-177.470,7.235,148.621
C01625=1173.731,238.312,-64.028,-177.467,7.238,148.621
C01626=1173.726,238.561,-64.055,-177.464,7.240,148.621
C01627=1173.722,238.809,-64.081,-177.461,7.243,148.621
C01628=1173.718,239.058,-64.107,-177.459,7.245,148.621
C01629=1173.713,239.307,-64.134,-177.456,7.247,148.620
C01630=1173.709,239.555,-64.160,-177.453,7.250,148.620
C01631=1173.704,239.804,-64.186,-177.451,7.253,148.620
C01632=1173.700,240.052,-64.213,-177.448,7.255,148.620
C01633=1173.695,240.301,-64.239,-177.446,7.257,148.620
C01634=1173.691,240.549,-64.265,-177.443,7.260,148.620
C01635=1173.686,240.797,-64.292,-177.440,7.262,148.619
C01636=1173.682,241.046,-64.318,-177.437,7.265,148.619
C01637=1173.677,241.295,-64.345,-177.435,7.268,148.619
C01638=1173.673,241.543,-64.371,-177.432,7.270,148.619
C01639=1173.668,241.792,-64.398,-177.429,7.273,148.619
C01640=1173.665,242.040,-64.425,-177.427,7.275,148.619
C01641=1173.660,242.289,-64.451,-177.424,7.278,148.619
C01642=1173.656,242.537,-64.477,-177.421,7.280,148.618
C01643=1173.651,242.786,-64.504,-177.419,7.283,148.618
C01644=1173.647,243.035,-64.530,-177.416,7.286,148.618
C01645=1173.642,243.283,-64.557,-177.414,7.287,148.618
C01646=1173.637,243.532,-64.584,-177.411,7.290,148.618
C01647=1173.633,243.780,-64.610,-177.408,7.293,148.618
C01648=1173.629,244.029,-64.637,-177.405,7.295,148.618
C01649=1173.625,244.277,-64.664,-177.403,7.298,148.617
C01650=1173.620,244.526,-64.691,-177.400,7.300,148.617
C01651=1173.615,244.775,-64.717,-177.397,7.303,148.617
C01652=1173.611,245.023,-64.743,-177.395,7.306,148.617
C01653=1173.606,245.271,-64.770,-177.392,7.308,148.617
C01654=1173.603,245.520,-64.797,-177.390,7.311,148.617
C01655=1173.598,245.768,-64.824,-177.386,7.314,148.617
C01656=1173.593,246.017,-64.851,-177.384,7.316,148.616
C01657=1173.589,246.265,-64.877,-177.381,7.319,148.616
C01658=1173.584,246.514,-64.904,-177.379,7.321,148.616
C01659=1173.580,246.763,-64.931,-177.376,7.323,148.616
C01660=1173.576,247.012,-64.958,-177.373,7.326,148.616
C01661=1173.572,247.260,-64.985,-177.371,7.329,148.616
C01662=1173.567,247.508,-65.012,-177.368,7.332,148.616
C01663=1173.562,247.757,-65.039,-177.365,7.334,148.616
C01664=1173.559,248.005,-65.065,-177.363,7.336,148.615
C01665=1173.554,248.253,-65.092,-177.360,7.339,148.615
C01666=1173.549,248.502,-65.120,-177.358,7.341,148.615
C01667=1173.545,248.750,-65.147,-177.355,7.344,148.615
C01668=1173.541,248.999,-65.173,-177.352,7.347,148.615
C01669=1173.536,249.247,-65.200,-177.350,7.349,148.615
C01670=1173.532,249.496,-65.228,-177.347,7.352,148.615
C01671=1173.527,249.745,-65.255,-177.344,7.355,148.614
C01672=1173.523,249.993,-65.282,-177.342,7.357,148.614
C01673=1173.519,250.242,-65.308,-177.339,7.360,148.614
C01674=1173.514,250.490,-65.335,-177.336,7.363,148.614
C01675=1173.509,250.739,-65.362,-177.334,7.365,148.614
C01676=1173.505,250.987,-65.389,-177.331,7.368,148.614
C01677=1173.501,251.236,-65.417,-177.328,7.371,148.614
C01678=1173.497,251.484,-65.443,-177.326,7.373,148.614
C01679=1173.492,251.733,-65.470,-177.323,7.376,148.614
C01680=1173.487,251.981,-65.497,-177.320,7.378,148.613
C01681=1173.483,252.230,-65.524,-177.318,7.380,148.613
C01682=1173.478,252.478,-65.552,-177.315,7.383,148.613
C01683=1173.474,252.727,-65.580,-177.312,7.386,148.613
C01684=1173.470,252.975,-65.607,-177.310,7.388,148.613
C01685=1173.465,253.224,-65.634,-177.307,7.391,148.613
C01686=1173.461,253.472,-65.660,-177.304,7.394,148.613
C01687=1173.457,253.720,-65.688,-177.302,7.396,148.613
C01688=1173.453,253.969,-65.715,-177.299,7.399,148.613
C01689=1173.448,254.218,-65.742,-177.296,7.402,148.613
C01690=1173.443,254.466,-65.770,-177.294,7.404,148.612
C01691=1173.439,254.714,-65.797,-177.291,7.407,148.612
C01692=1173.435,254.963,-65.825,-177.288,7.410,148.612
C01693=1173.430,255.212,-65.852,-177.286,7.412,148.612
C01694=1173.426,255.460,-65.880,-177.283,7.415,148.612
C01695=1173.421,255.708,-65.907,-177.281,7.418,148.612
C01696=1173.417,255.957,-65.934,-177.278,7.420,148.612
C01697=1173.413,256.205,-65.962,-177.275,7.423,148.611
C01698=1173.408,256.454,-65.989,-177.273,7.426,148.611
C01699=1173.404,256.702,-66.016,-177.270,7.428,148.611
C01700=1173.400,256.951,-66.044,-177.268,7.431,148.611
C01701=1173.395,257.199,-66.071,-177.265,7.434,148.611
C01702=1173.391,257.447,-66.099,-177.263,7.436,148.611
C01703=1173.386,257.696,-66.126,-177.259,7.439,148.611
C01704=1173.382,257.945,-66.153,-177.257,7.442,148.611
C01705=1173.378,258.193,-66.181,-177.254,7.445,148.611
C01706=1173.373,258.441,-66.208,-177.252,7.447,148.611
C01707=1173.369,258.690,-66.236,-177.249,7.450,148.611
C01708=1173.364,258.939,-66.264,-177.246,7.453,148.611
C01709=1173.360,259.186,-66.292,-177.244,7.455,148.610
C01710=1173.356,259.436,-66.319,-177.241,7.457,148.610
C01711=1173.351,259.684,-66.347,-177.238,7.460,148.610
C01712=1173.347,259.932,-66.374,-177.235,7.463,148.610
C01713=1173.343,260.181,-66.402,-177.233,7.465,148.610
C01714=1173.338,260.428,-66.430,-177.230,7.468,148.610
C01715=1173.334,260.677,-66.457,-177.228,7.471,148.610
C01716=1173.329,260.926,-66.486,-177.226,7.474,148.610
C01717=1173.325,261.174,-66.513,-177.223,7.477,148.610
C01718=1173.320,261.422,-66.541,-177.220,7.479,148.610
C01719=1173.317,261.671,-66.569,-177.217,7.482,148.609
C01720=1173.311,261.943,-66.599,-177.214,7.485,148.609
C01721=1173.307,262.217,-66.630,-177.211,7.488,148.609
C01722=1173.302,262.490,-66.660,-177.209,7.491,148.609
C01723=1173.297,262.763,-66.691,-177.206,7.494,148.609
C01724=1173.293,263.011,-66.719,-177.203,7.497,148.609
C01725=1173.288,263.260,-66.746,-177.200,7.500,148.609
C01726=1173.284,263.509,-66.775,-177.198,7.502,148.609
C01727=1173.279,263.757,-66.803,-177.195,7.505,148.609
C01728=1173.275,264.004,-66.830,-177.192,7.508,148.609
C01729=1173.271,264.254,-66.858,-177.190,7.510,148.609
C01730=1173.266,264.502,-66.886,-177.187,7.513,148.609
C01731=1173.262,264.750,-66.914,-177.185,7.516,148.608
C01732=1173.258,264.998,-66.942,-177.182,7.519,148.608
C01733=1173.253,265.248,-66.970,-177.180,7.521,148.608
C01734=1173.249,265.496,-66.998,-177.177,7.524,148.608
C01735=1173.244,265.744,-67.026,-177.174,7.527,148.608
C01736=1173.240,265.992,-67.054,-177.171,7.530,148.608
C01737=1173.236,266.240,-67.082,-177.169,7.532,148.608
C01738=1173.232,266.489,-67.110,-177.167,7.535,148.608
C01739=1173.227,266.737,-67.139,-177.164,7.538,148.608
C01740=1173.223,266.986,-67.167,-177.161,7.541,148.608
C01741=1173.218,267.234,-67.194,-177.158,7.544,148.608
C01742=1173.214,267.483,-67.223,-177.156,7.546,148.608
C01743=1173.209,267.731,-67.250,-177.153,7.549,148.608
C01744=1173.205,267.980,-67.279,-177.150,7.552,148.607
C01745=1173.201,268.228,-67.307,-177.147,7.555,148.607
C01746=1173.197,268.476,-67.335,-177.145,7.557,148.607
C01747=1173.192,268.724,-67.363,-177.143,7.560,148.607
C01748=1173.188,268.973,-67.392,-177.140,7.563,148.607
C01749=1173.183,269.221,-67.420,-177.137,7.566,148.607
C01750=1173.179,269.470,-67.448,-177.135,7.568,148.607
C01751=1173.174,269.718,-67.476,-177.132,7.571,148.607
C01752=1173.170,269.967,-67.505,-177.129,7.574,148.607
C01753=1173.166,270.214,-67.533,-177.127,7.577,148.607
C01754=1173.162,270.463,-67.562,-177.124,7.580,148.607
C01755=1173.157,270.711,-67.590,-177.122,7.582,148.607
C01756=1173.153,270.959,-67.618,-177.119,7.585,148.607
C01757=1173.149,271.208,-67.646,-177.116,7.588,148.607
C01758=1173.144,271.456,-67.675,-177.113,7.591,148.607
C01759=1173.140,271.705,-67.703,-177.111,7.594,148.607
C01760=1173.135,271.953,-67.731,-177.109,7.596,148.607
C01761=1173.131,272.201,-67.761,-177.106,7.599,148.607
C01762=1173.127,272.450,-67.789,-177.103,7.602,148.606
C01763=1173.122,272.698,-67.817,-177.100,7.605,148.606
C01764=1173.119,272.947,-67.845,-177.098,7.607,148.606
C01765=1173.114,273.194,-67.875,-177.095,7.610,148.606
C01766=1173.110,273.443,-67.903,-177.093,7.613,148.606
C01767=1173.106,273.692,-67.931,-177.090,7.616,148.606
C01768=1173.100,273.940,-67.960,-177.087,7.619,148.606
C01769=1173.097,274.188,-67.989,-177.085,7.621,148.606
C01770=1173.092,274.436,-68.017,-177.082,7.624,148.606
C01771=1173.088,274.684,-68.045,-177.080,7.627,148.606
C01772=1173.084,274.933,-68.075,-177.077,7.630,148.606
C01773=1173.079,275.181,-68.103,-177.075,7.633,148.606
C01774=1173.075,275.430,-68.131,-177.072,7.636,148.606
C01775=1173.071,275.678,-68.161,-177.070,7.638,148.606
C01776=1173.066,275.926,-68.189,-177.067,7.641,148.606
C01777=1173.062,276.175,-68.217,-177.064,7.644,148.606
C01778=1173.058,276.423,-68.247,-177.061,7.647,148.606
C01779=1173.053,276.671,-68.275,-177.059,7.650,148.606
C01780=1173.049,276.919,-68.304,-177.056,7.652,148.606
C01781=1173.045,277.168,-68.333,-177.054,7.655,148.606
C01782=1173.040,277.416,-68.361,-177.051,7.658,148.606
C01783=1173.036,277.664,-68.390,-177.048,7.661,148.606
C01784=1173.032,277.913,-68.418,-177.045,7.664,148.606
C01785=1173.028,278.161,-68.448,-177.043,7.667,148.606
C01786=1173.023,278.409,-68.476,-177.041,7.669,148.605
C01787=1173.019,278.657,-68.505,-177.038,7.672,148.605
C01788=1173.015,278.906,-68.534,-177.035,7.675,148.605
C01789=1173.011,279.154,-68.563,-177.032,7.678,148.605
C01790=1173.006,279.402,-68.592,-177.030,7.682,148.605
C01791=1173.002,279.651,-68.621,-177.027,7.685,148.605
C01792=1172.998,279.899,-68.650,-177.025,7.687,148.605
C01793=1172.993,280.147,-68.678,-177.022,7.690,148.605
C01794=1172.989,280.395,-68.708,-177.020,7.693,148.605
C01795=1172.984,280.644,-68.737,-177.017,7.696,148.605
C01796=1172.981,280.892,-68.765,-177.014,7.699,148.605
C01797=1172.976,281.140,-68.795,-177.011,7.702,148.605
C01798=1172.972,281.388,-68.824,-177.009,7.704,148.605
C01799=1172.967,281.637,-68.853,-177.007,7.707,148.605
C01800=1172.963,281.885,-68.882,-177.004,7.710,148.605
C01801=1172.959,282.133,-68.912,-177.002,7.713,148.605
C01802=1172.954,282.382,-68.940,-176.999,7.716,148.605
C01803=1172.950,282.630,-68.969,-176.996,7.719,148.605
C01804=1172.946,282.878,-68.998,-176.993,7.722,148.605
C01805=1172.942,283.126,-69.028,-176.991,7.724,148.605
C01806=1172.937,283.375,-69.057,-176.988,7.727,148.605
C01807=1172.933,283.623,-69.086,-176.986,7.730,148.605
C01808=1172.928,283.871,-69.115,-176.983,7.733,148.605
C01809=1172.924,284.119,-69.145,-176.981,7.736,148.605
C01810=1172.920,284.367,-69.174,-176.978,7.739,148.605
C01811=1172.916,284.616,-69.203,-176.975,7.742,148.605
C01812=1172.911,284.864,-69.232,-176.972,7.745,148.605
C01813=1172.907,285.112,-69.261,-176.970,7.747,148.605
C01814=1172.902,285.360,-69.291,-176.968,7.750,148.605
C01815=1172.898,285.609,-69.320,-176.965,7.753,148.605
C01816=1172.894,285.857,-69.350,-176.962,7.757,148.605
C01817=1172.890,286.105,-69.379,-176.960,7.760,148.605
C01818=1172.886,286.353,-69.409,-176.957,7.763,148.605
C01819=1172.881,286.602,-69.437,-176.954,7.766,148.605
C01820=1172.877,286.851,-69.467,-176.952,7.768,148.605
C01821=1172.872,287.098,-69.496,-176.949,7.771,148.605
C01822=1172.868,287.346,-69.525,-176.947,7.774,148.605
C01823=1172.864,287.595,-69.555,-176.944,7.777,148.605
C01824=1172.859,287.869,-69.588,-176.942,7.780,148.605
C01825=1172.854,288.145,-69.621,-176.938,7.784,148.605
C01826=1172.850,288.419,-69.653,-176.936,7.787,148.605
